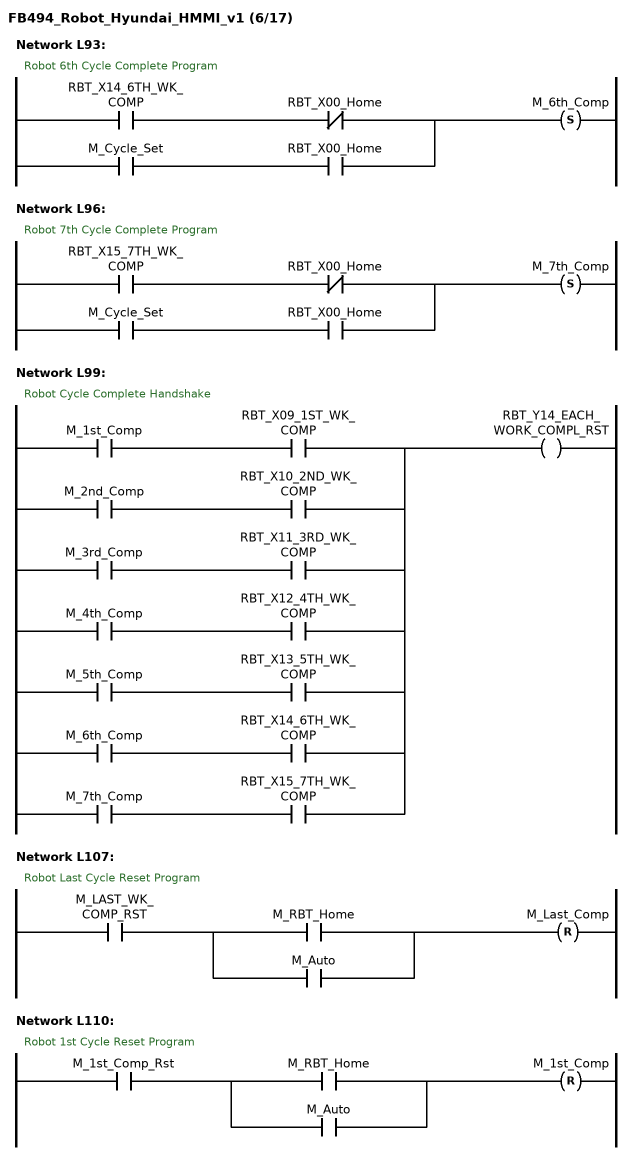
(* [picture p24: FB494_Robot_Hyundai_HMMI_v1 rungs L93-L110] *)
(* Robot 6th Cycle Complete Program *)
(* Rung L93 *)
IF (RBT_X14_6TH_WK_COMP AND NOT RBT_X00_Home) OR (M_Cycle_Set AND RBT_X00_Home) THEN
    M_6th_Comp := TRUE;
END_IF;
(* Robot 7th Cycle Complete Program *)
(* Rung L96 *)
IF (RBT_X15_7TH_WK_COMP AND NOT RBT_X00_Home) OR (M_Cycle_Set AND RBT_X00_Home) THEN
    M_7th_Comp := TRUE;
END_IF;
(* Robot Cycle Complete Handshake *)
(* Rung L99 *)
RBT_Y14_EACH_WORK_COMPL_RST := (M_1st_Comp AND RBT_X09_1ST_WK_COMP) OR (M_2nd_Comp AND RBT_X10_2ND_WK_COMP) OR (M_3rd_Comp AND RBT_X11_3RD_WK_COMP) OR (M_4th_Comp AND RBT_X12_4TH_WK_COMP) OR (M_5th_Comp AND RBT_X13_5TH_WK_COMP) OR (M_6th_Comp AND RBT_X14_6TH_WK_COMP) OR (M_7th_Comp AND RBT_X15_7TH_WK_COMP);
(* Robot Last Cycle Reset Program *)
(* Rung L107 *)
IF M_LAST_WK_COMP_RST AND (M_RBT_Home OR M_Auto) THEN M_Last_Comp := FALSE; END_IF;
(* Robot 1st Cycle Reset Program *)
(* Rung L110 *)
IF M_1st_Comp_Rst AND (M_RBT_Home OR M_Auto) THEN M_1st_Comp := FALSE; END_IF;

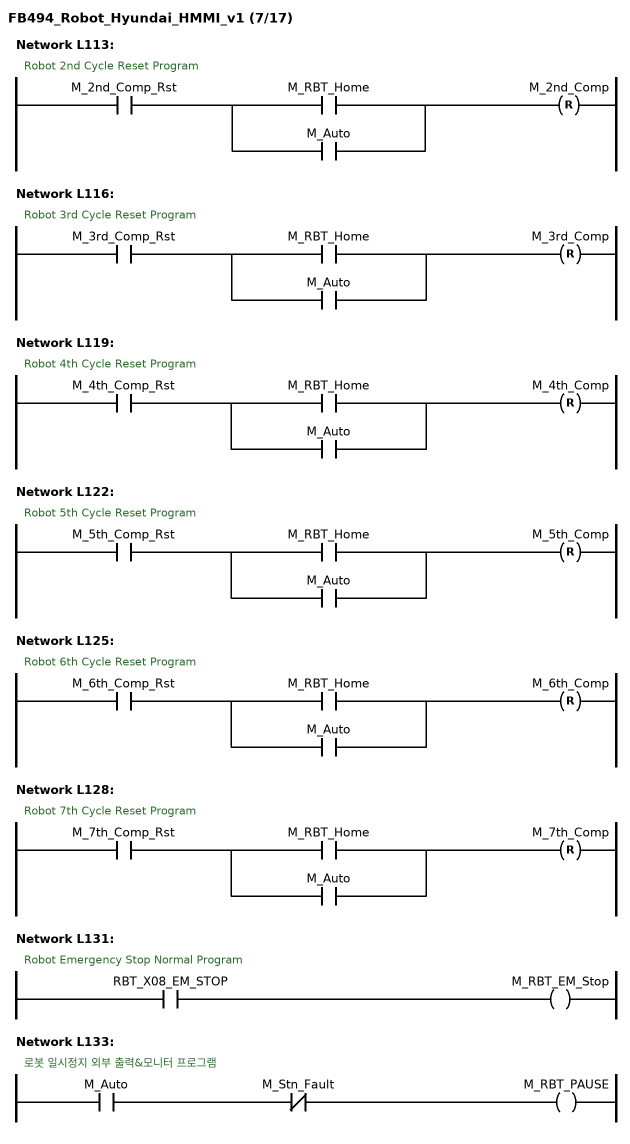
(* Robot 2nd Cycle Reset Program *)
(* Rung L113 *)
IF M_2nd_Comp_Rst AND (M_RBT_Home OR M_Auto) THEN M_2nd_Comp := FALSE; END_IF;
(* Robot 3rd Cycle Reset Program *)
(* Rung L116 *)
IF M_3rd_Comp_Rst AND (M_RBT_Home OR M_Auto) THEN M_3rd_Comp := FALSE; END_IF;
(* Robot 4th Cycle Reset Program *)
(* Rung L119 *)
IF M_4th_Comp_Rst AND (M_RBT_Home OR M_Auto) THEN M_4th_Comp := FALSE; END_IF;
(* Robot 5th Cycle Reset Program *)
(* Rung L122 *)
IF M_5th_Comp_Rst AND (M_RBT_Home OR M_Auto) THEN M_5th_Comp := FALSE; END_IF;
(* Robot 6th Cycle Reset Program *)
(* Rung L125 *)
IF M_6th_Comp_Rst AND (M_RBT_Home OR M_Auto) THEN M_6th_Comp := FALSE; END_IF;
(* Robot 7th Cycle Reset Program *)
(* Rung L128 *)
IF M_7th_Comp_Rst AND (M_RBT_Home OR M_Auto) THEN M_7th_Comp := FALSE; END_IF;
(* Robot Emergency Stop Normal Program *)
(* Rung L131 *)
M_RBT_EM_Stop := RBT_X08_EM_STOP;
(* 로봇 일시정지 외부 출력&모니터 프로그램 *)
(* Rung L133 *)
M_RBT_PAUSE := M_Auto AND NOT M_Stn_Fault;

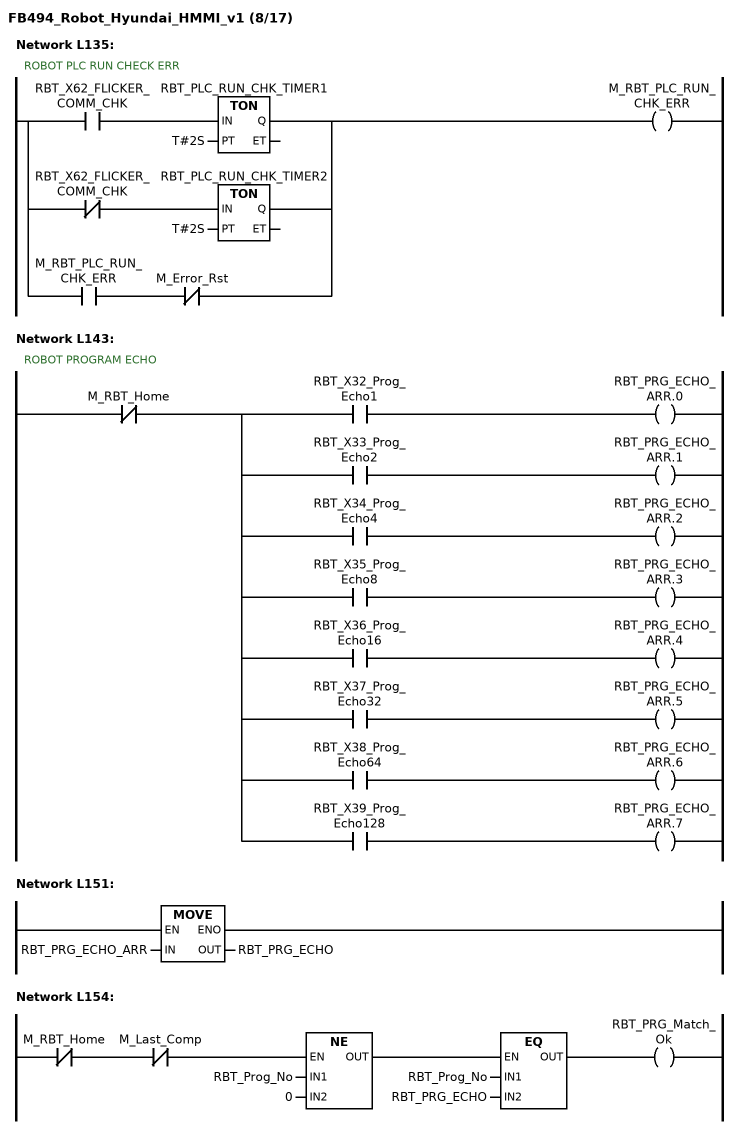
(* ROBOT PLC RUN CHECK ERR *)
(* Rung L135 *)
RBT_PLC_RUN_CHK_TIMER1(IN := RBT_X62_FLICKER_COMM_CHK, PT := T#2S);
RBT_PLC_RUN_CHK_TIMER2(IN := NOT RBT_X62_FLICKER_COMM_CHK, PT := T#2S);
M_RBT_PLC_RUN_CHK_ERR := RBT_PLC_RUN_CHK_TIMER1.Q OR RBT_PLC_RUN_CHK_TIMER2.Q OR (M_RBT_PLC_RUN_CHK_ERR AND NOT M_Error_Rst);
(* ROBOT PROGRAM ECHO *)
(* Rung L143 *)
RBT_PRG_ECHO_ARR.0 := NOT M_RBT_Home AND RBT_X32_Prog_Echo1;
RBT_PRG_ECHO_ARR.1 := NOT M_RBT_Home AND RBT_X33_Prog_Echo2;
RBT_PRG_ECHO_ARR.2 := NOT M_RBT_Home AND RBT_X34_Prog_Echo4;
RBT_PRG_ECHO_ARR.3 := NOT M_RBT_Home AND RBT_X35_Prog_Echo8;
RBT_PRG_ECHO_ARR.4 := NOT M_RBT_Home AND RBT_X36_Prog_Echo16;
RBT_PRG_ECHO_ARR.5 := NOT M_RBT_Home AND RBT_X37_Prog_Echo32;
RBT_PRG_ECHO_ARR.6 := NOT M_RBT_Home AND RBT_X38_Prog_Echo64;
RBT_PRG_ECHO_ARR.7 := NOT M_RBT_Home AND RBT_X39_Prog_Echo128;
(* Rung L151 *)
RBT_PRG_ECHO := RBT_PRG_ECHO_ARR;
(* Rung L154 *)
IF NOT M_RBT_Home AND NOT M_Last_Comp THEN _t1 := RBT_Prog_No <> 0; END_IF;
IF _t1 THEN _t2 := RBT_Prog_No = RBT_PRG_ECHO; END_IF;
RBT_PRG_Match_Ok := _t2;

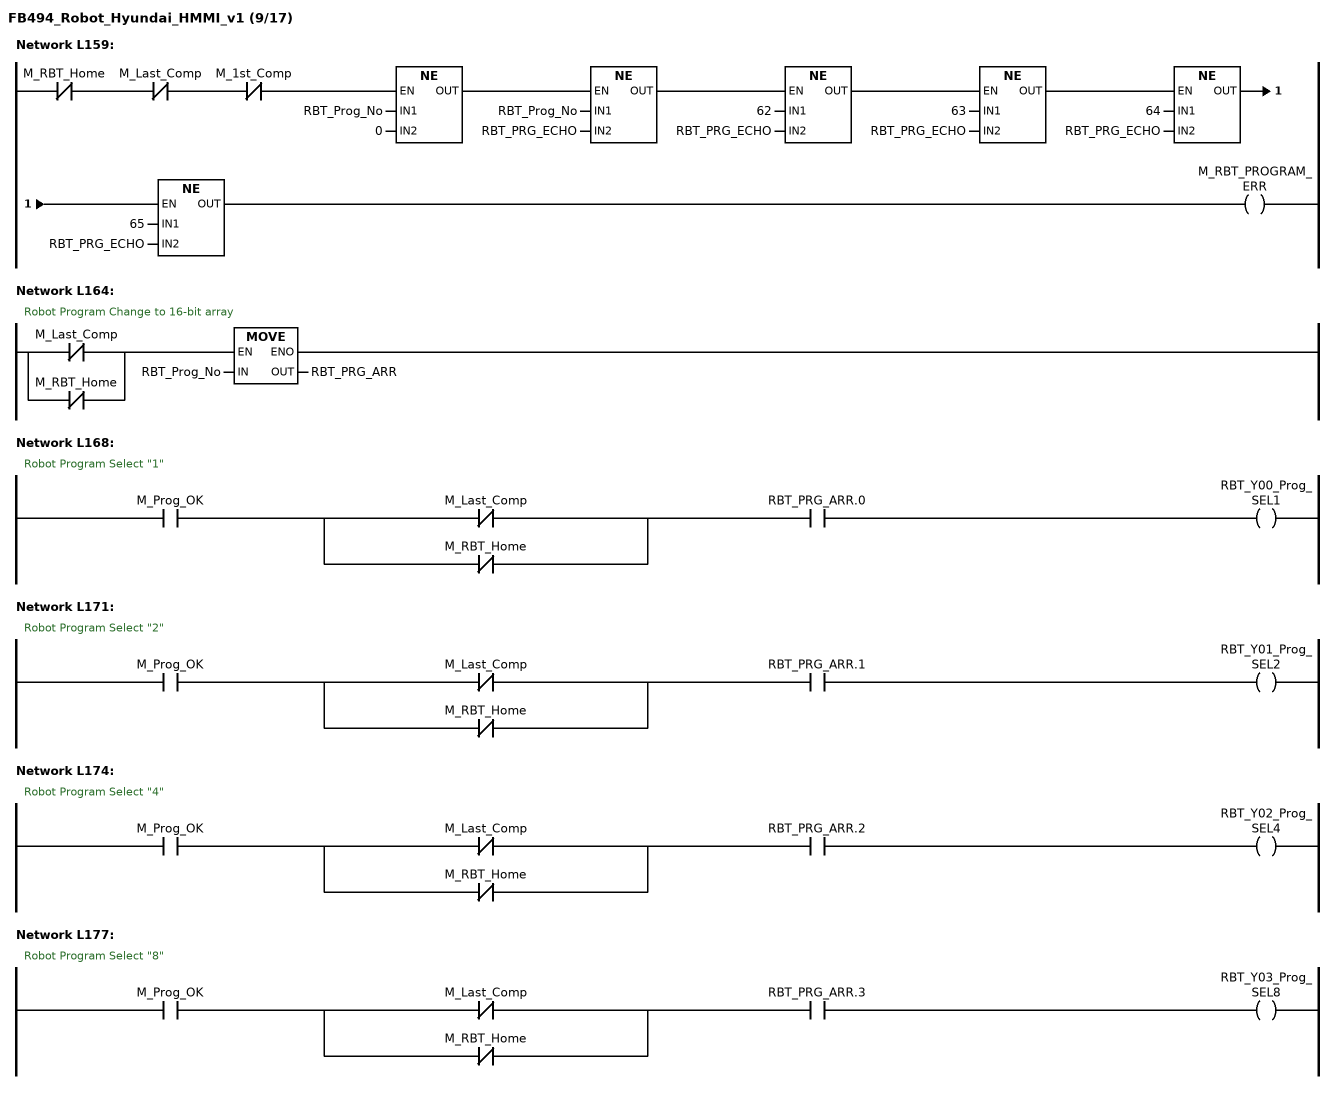
(* Rung L159 *)
IF NOT M_RBT_Home AND NOT M_Last_Comp AND NOT M_1st_Comp THEN _t3 := RBT_Prog_No <> 0; END_IF;
IF _t3 THEN _t4 := RBT_Prog_No <> RBT_PRG_ECHO; END_IF;
IF _t4 THEN _t5 := 62 <> RBT_PRG_ECHO; END_IF;
IF _t5 THEN _t6 := 63 <> RBT_PRG_ECHO; END_IF;
IF _t6 THEN _t7 := 64 <> RBT_PRG_ECHO; END_IF;
IF _t7 THEN _t8 := 65 <> RBT_PRG_ECHO; END_IF;
M_RBT_PROGRAM_ERR := _t8;
(* Robot Program Change to 16-bit array *)
(* Rung L164 *)
IF NOT M_Last_Comp OR NOT M_RBT_Home THEN RBT_PRG_ARR := RBT_Prog_No; END_IF;
(* Robot Program Select "1" *)
(* Rung L168 *)
RBT_Y00_Prog_SEL1 := M_Prog_OK AND (NOT M_Last_Comp OR NOT M_RBT_Home) AND RBT_PRG_ARR.0;
(* Robot Program Select "2" *)
(* Rung L171 *)
RBT_Y01_Prog_SEL2 := M_Prog_OK AND (NOT M_Last_Comp OR NOT M_RBT_Home) AND RBT_PRG_ARR.1;
(* Robot Program Select "4" *)
(* Rung L174 *)
RBT_Y02_Prog_SEL4 := M_Prog_OK AND (NOT M_Last_Comp OR NOT M_RBT_Home) AND RBT_PRG_ARR.2;
(* Robot Program Select "8" *)
(* Rung L177 *)
RBT_Y03_Prog_SEL8 := M_Prog_OK AND (NOT M_Last_Comp OR NOT M_RBT_Home) AND RBT_PRG_ARR.3;

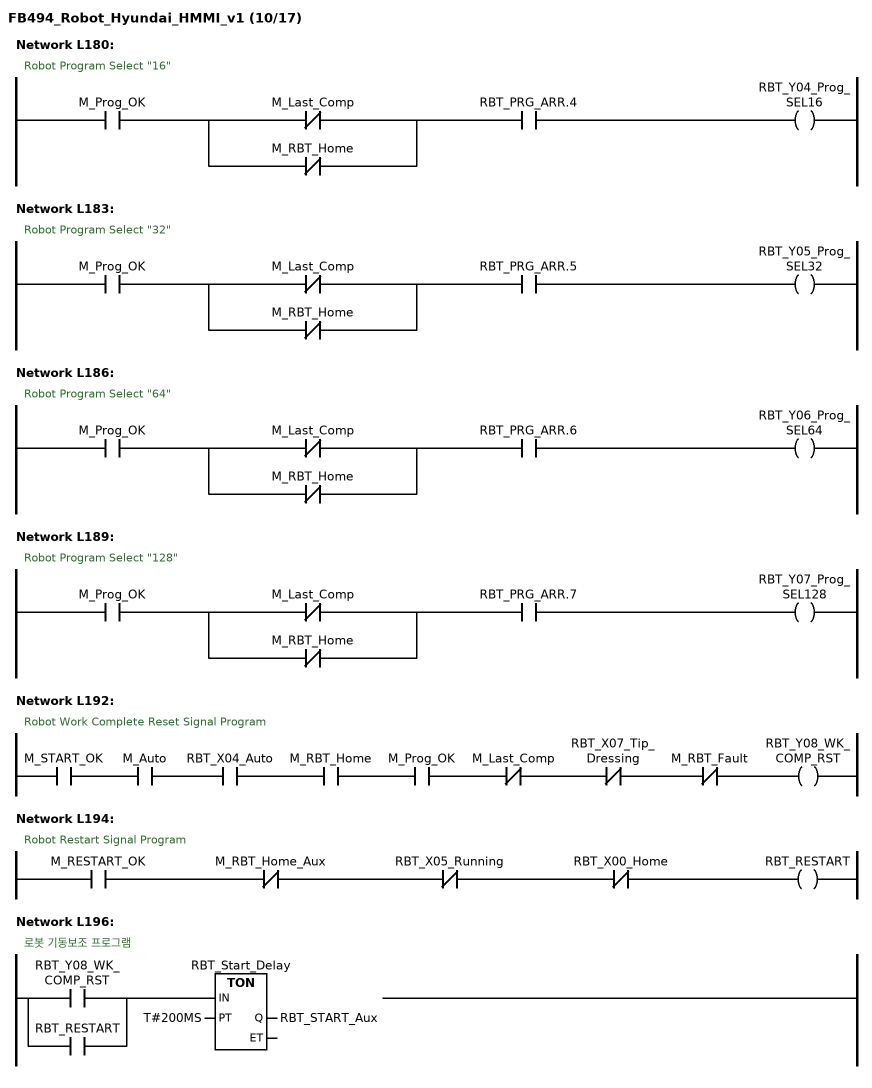
(* Robot Program Select "16" *)
(* Rung L180 *)
RBT_Y04_Prog_SEL16 := M_Prog_OK AND (NOT M_Last_Comp OR NOT M_RBT_Home) AND RBT_PRG_ARR.4;
(* Robot Program Select "32" *)
(* Rung L183 *)
RBT_Y05_Prog_SEL32 := M_Prog_OK AND (NOT M_Last_Comp OR NOT M_RBT_Home) AND RBT_PRG_ARR.5;
(* Robot Program Select "64" *)
(* Rung L186 *)
RBT_Y06_Prog_SEL64 := M_Prog_OK AND (NOT M_Last_Comp OR NOT M_RBT_Home) AND RBT_PRG_ARR.6;
(* Robot Program Select "128" *)
(* Rung L189 *)
RBT_Y07_Prog_SEL128 := M_Prog_OK AND (NOT M_Last_Comp OR NOT M_RBT_Home) AND RBT_PRG_ARR.7;
(* Robot Work Complete Reset Signal Program *)
(* Rung L192 *)
RBT_Y08_WK_COMP_RST := M_START_OK AND M_Auto AND RBT_X04_Auto AND M_RBT_Home AND M_Prog_OK AND NOT M_Last_Comp AND NOT RBT_X07_Tip_Dressing AND NOT M_RBT_Fault;
(* Robot Restart Signal Program *)
(* Rung L194 *)
RBT_RESTART := M_RESTART_OK AND NOT M_RBT_Home_Aux AND NOT RBT_X05_Running AND NOT RBT_X00_Home;
(* 로봇 기동보조 프로그램 *)
(* Rung L196 *)
RBT_Start_Delay(IN := RBT_Y08_WK_COMP_RST OR RBT_RESTART, PT := T#200MS, Q => RBT_START_Aux);

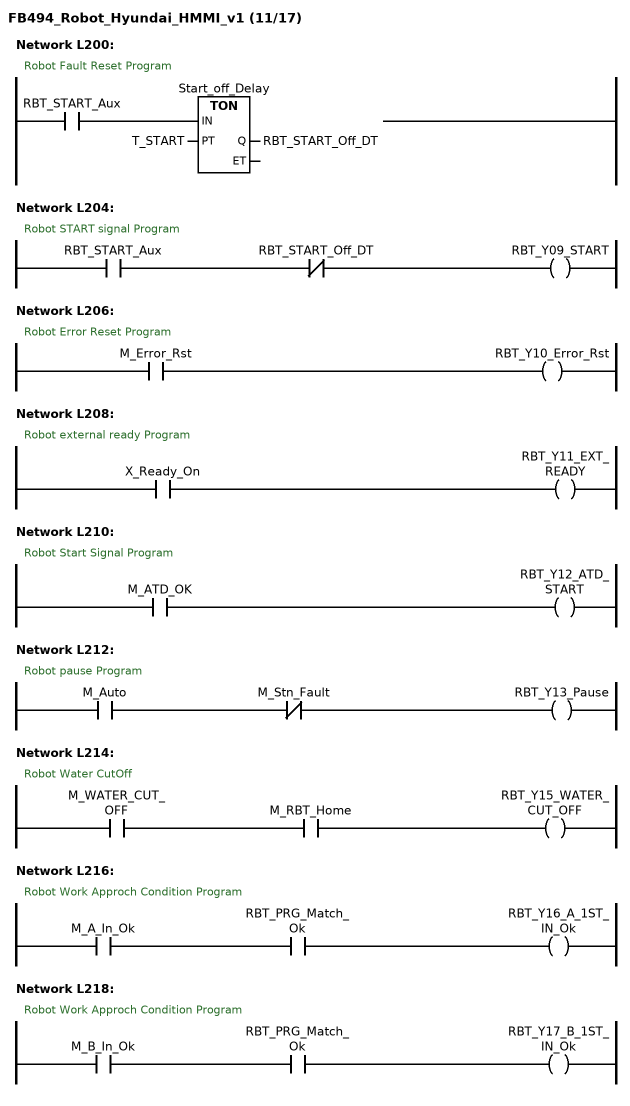
(* Robot Fault Reset Program *)
(* Rung L200 *)
Start_off_Delay(IN := RBT_START_Aux, PT := T_START, Q => RBT_START_Off_DT);
(* Robot START signal Program *)
(* Rung L204 *)
RBT_Y09_START := RBT_START_Aux AND NOT RBT_START_Off_DT;
(* Robot Error Reset Program *)
(* Rung L206 *)
RBT_Y10_Error_Rst := M_Error_Rst;
(* Robot external ready Program *)
(* Rung L208 *)
RBT_Y11_EXT_READY := X_Ready_On;
(* Robot Start Signal Program *)
(* Rung L210 *)
RBT_Y12_ATD_START := M_ATD_OK;
(* Robot pause Program *)
(* Rung L212 *)
RBT_Y13_Pause := M_Auto AND NOT M_Stn_Fault;
(* Robot Water CutOff *)
(* Rung L214 *)
RBT_Y15_WATER_CUT_OFF := M_WATER_CUT_OFF AND M_RBT_Home;
(* Robot Work Approch Condition Program *)
(* Rung L216 *)
RBT_Y16_A_1ST_IN_Ok := M_A_In_Ok AND RBT_PRG_Match_Ok;
(* Robot Work Approch Condition Program *)
(* Rung L218 *)
RBT_Y17_B_1ST_IN_Ok := M_B_In_Ok AND RBT_PRG_Match_Ok;

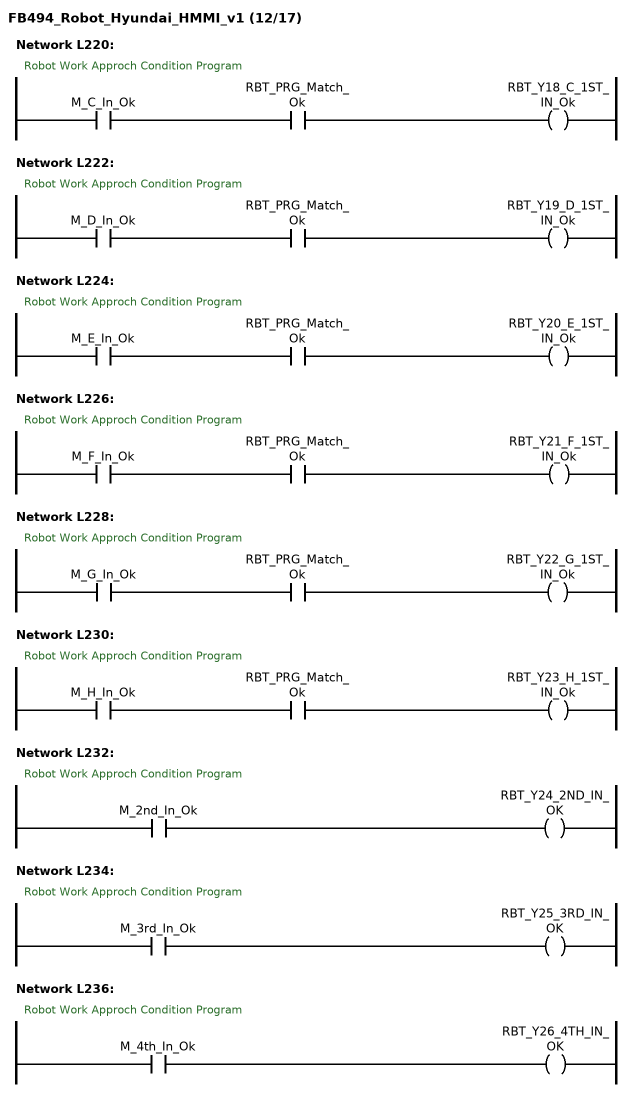
(* Robot Work Approch Condition Program *)
(* Rung L220 *)
RBT_Y18_C_1ST_IN_Ok := M_C_In_Ok AND RBT_PRG_Match_Ok;
(* Robot Work Approch Condition Program *)
(* Rung L222 *)
RBT_Y19_D_1ST_IN_Ok := M_D_In_Ok AND RBT_PRG_Match_Ok;
(* Robot Work Approch Condition Program *)
(* Rung L224 *)
RBT_Y20_E_1ST_IN_Ok := M_E_In_Ok AND RBT_PRG_Match_Ok;
(* Robot Work Approch Condition Program *)
(* Rung L226 *)
RBT_Y21_F_1ST_IN_Ok := M_F_In_Ok AND RBT_PRG_Match_Ok;
(* Robot Work Approch Condition Program *)
(* Rung L228 *)
RBT_Y22_G_1ST_IN_Ok := M_G_In_Ok AND RBT_PRG_Match_Ok;
(* Robot Work Approch Condition Program *)
(* Rung L230 *)
RBT_Y23_H_1ST_IN_Ok := M_H_In_Ok AND RBT_PRG_Match_Ok;
(* Robot Work Approch Condition Program *)
(* Rung L232 *)
RBT_Y24_2ND_IN_OK := M_2nd_In_Ok;
(* Robot Work Approch Condition Program *)
(* Rung L234 *)
RBT_Y25_3RD_IN_OK := M_3rd_In_Ok;
(* Robot Work Approch Condition Program *)
(* Rung L236 *)
RBT_Y26_4TH_IN_OK := M_4th_In_Ok;

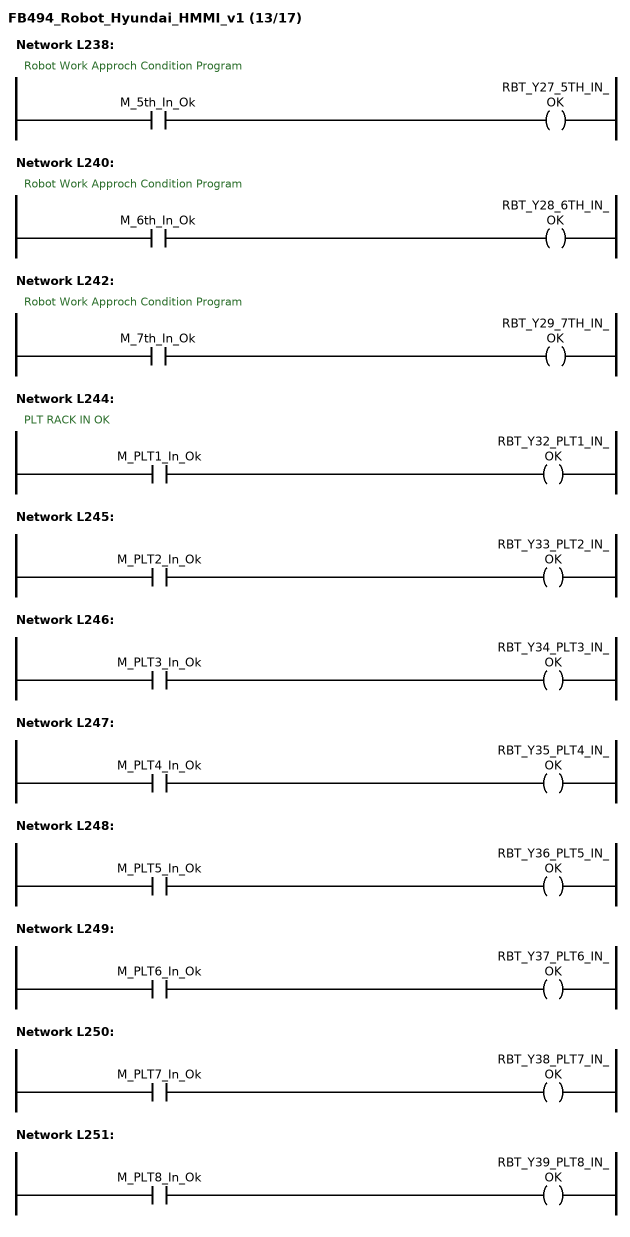
(* Robot Work Approch Condition Program *)
(* Rung L238 *)
RBT_Y27_5TH_IN_OK := M_5th_In_Ok;
(* Robot Work Approch Condition Program *)
(* Rung L240 *)
RBT_Y28_6TH_IN_OK := M_6th_In_Ok;
(* Robot Work Approch Condition Program *)
(* Rung L242 *)
RBT_Y29_7TH_IN_OK := M_7th_In_Ok;
(* PLT RACK IN OK *)
(* Rung L244 *)
RBT_Y32_PLT1_IN_OK := M_PLT1_In_Ok;
(* Rung L245 *)
RBT_Y33_PLT2_IN_OK := M_PLT2_In_Ok;
(* Rung L246 *)
RBT_Y34_PLT3_IN_OK := M_PLT3_In_Ok;
(* Rung L247 *)
RBT_Y35_PLT4_IN_OK := M_PLT4_In_Ok;
(* Rung L248 *)
RBT_Y36_PLT5_IN_OK := M_PLT5_In_Ok;
(* Rung L249 *)
RBT_Y37_PLT6_IN_OK := M_PLT6_In_Ok;
(* Rung L250 *)
RBT_Y38_PLT7_IN_OK := M_PLT7_In_Ok;
(* Rung L251 *)
RBT_Y39_PLT8_IN_OK := M_PLT8_In_Ok;

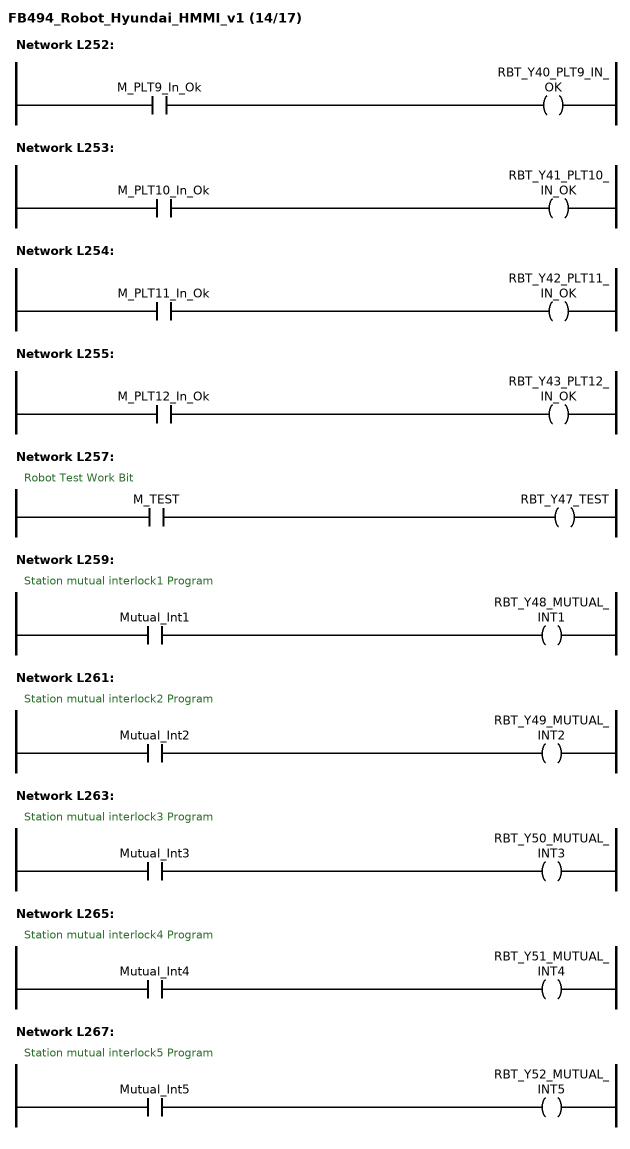
(* Rung L252 *)
RBT_Y40_PLT9_IN_OK := M_PLT9_In_Ok;
(* Rung L253 *)
RBT_Y41_PLT10_IN_OK := M_PLT10_In_Ok;
(* Rung L254 *)
RBT_Y42_PLT11_IN_OK := M_PLT11_In_Ok;
(* Rung L255 *)
RBT_Y43_PLT12_IN_OK := M_PLT12_In_Ok;
(* Robot Test Work Bit *)
(* Rung L257 *)
RBT_Y47_TEST := M_TEST;
(* Station mutual interlock1 Program *)
(* Rung L259 *)
RBT_Y48_MUTUAL_INT1 := Mutual_Int1;
(* Station mutual interlock2 Program *)
(* Rung L261 *)
RBT_Y49_MUTUAL_INT2 := Mutual_Int2;
(* Station mutual interlock3 Program *)
(* Rung L263 *)
RBT_Y50_MUTUAL_INT3 := Mutual_Int3;
(* Station mutual interlock4 Program *)
(* Rung L265 *)
RBT_Y51_MUTUAL_INT4 := Mutual_Int4;
(* Station mutual interlock5 Program *)
(* Rung L267 *)
RBT_Y52_MUTUAL_INT5 := Mutual_Int5;

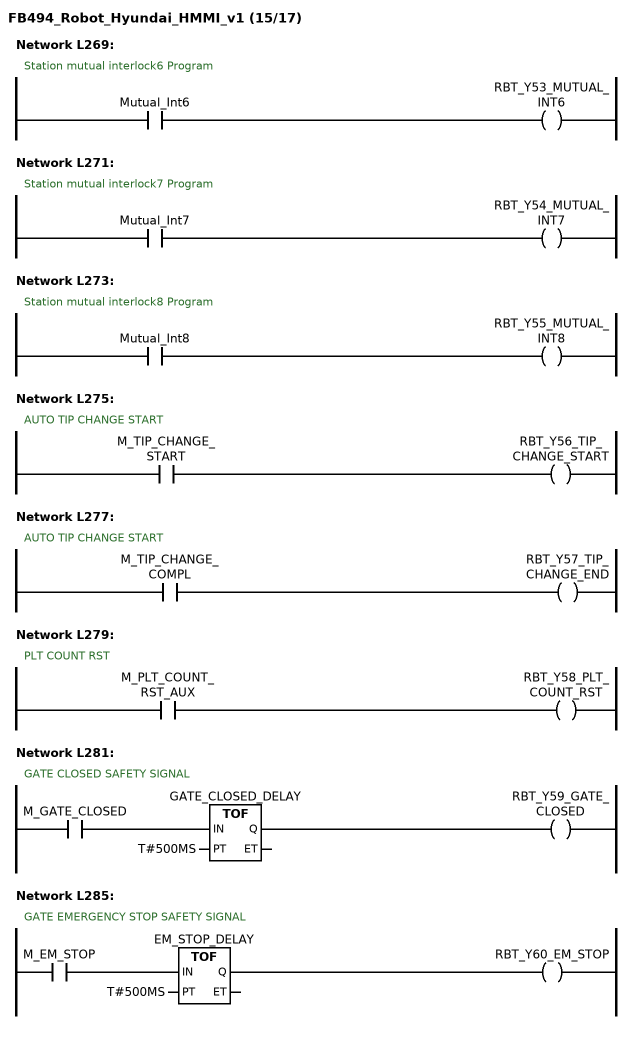
(* Station mutual interlock6 Program *)
(* Rung L269 *)
RBT_Y53_MUTUAL_INT6 := Mutual_Int6;
(* Station mutual interlock7 Program *)
(* Rung L271 *)
RBT_Y54_MUTUAL_INT7 := Mutual_Int7;
(* Station mutual interlock8 Program *)
(* Rung L273 *)
RBT_Y55_MUTUAL_INT8 := Mutual_Int8;
(* AUTO TIP CHANGE START *)
(* Rung L275 *)
RBT_Y56_TIP_CHANGE_START := M_TIP_CHANGE_START;
(* AUTO TIP CHANGE START *)
(* Rung L277 *)
RBT_Y57_TIP_CHANGE_END := M_TIP_CHANGE_COMPL;
(* PLT COUNT RST *)
(* Rung L279 *)
RBT_Y58_PLT_COUNT_RST := M_PLT_COUNT_RST_AUX;
(* GATE CLOSED SAFETY SIGNAL *)
(* Rung L281 *)
GATE_CLOSED_DELAY(IN := M_GATE_CLOSED, PT := T#500MS);
RBT_Y59_GATE_CLOSED := GATE_CLOSED_DELAY.Q;
(* GATE EMERGENCY STOP SAFETY SIGNAL *)
(* Rung L285 *)
EM_STOP_DELAY(IN := M_EM_STOP, PT := T#500MS);
RBT_Y60_EM_STOP := EM_STOP_DELAY.Q;

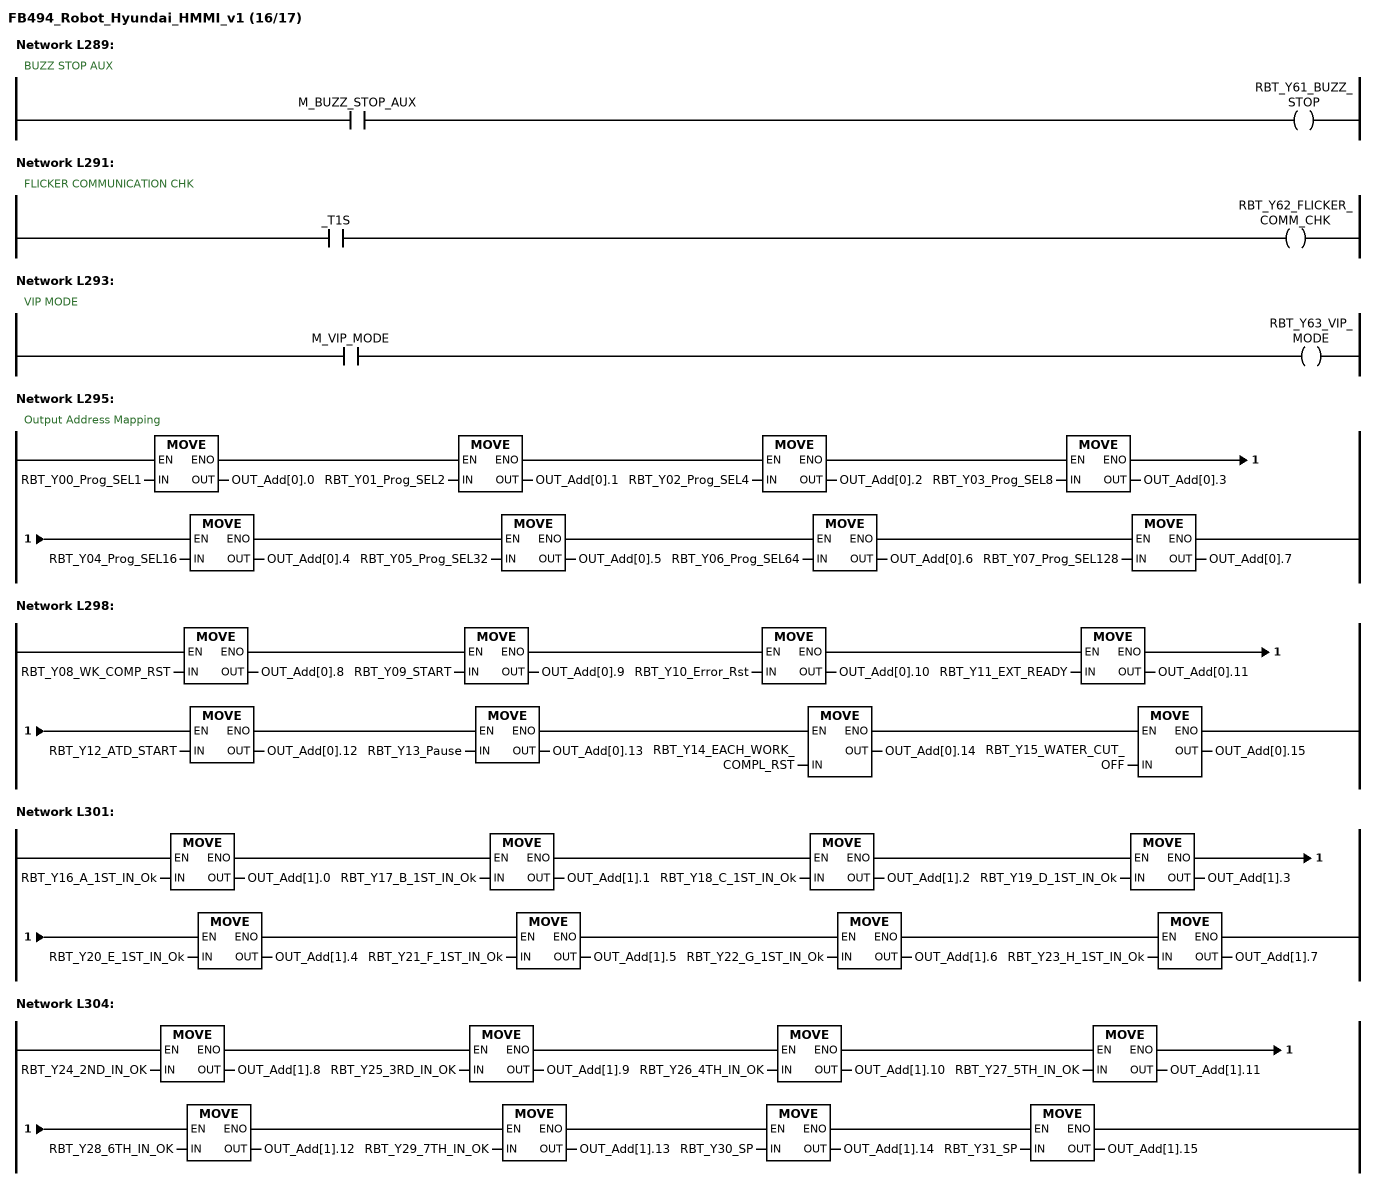
(* BUZZ STOP AUX *)
(* Rung L289 *)
RBT_Y61_BUZZ_STOP := M_BUZZ_STOP_AUX;
(* FLICKER COMMUNICATION CHK *)
(* Rung L291 *)
RBT_Y62_FLICKER_COMM_CHK := _T1S;
(* VIP MODE *)
(* Rung L293 *)
RBT_Y63_VIP_MODE := M_VIP_MODE;
(* Output Address Mapping *)
(* Rung L295 *)
OUT_Add[0].0 := RBT_Y00_Prog_SEL1;
OUT_Add[0].1 := RBT_Y01_Prog_SEL2;
OUT_Add[0].2 := RBT_Y02_Prog_SEL4;
OUT_Add[0].3 := RBT_Y03_Prog_SEL8;
OUT_Add[0].4 := RBT_Y04_Prog_SEL16;
OUT_Add[0].5 := RBT_Y05_Prog_SEL32;
OUT_Add[0].6 := RBT_Y06_Prog_SEL64;
OUT_Add[0].7 := RBT_Y07_Prog_SEL128;
(* Rung L298 *)
OUT_Add[0].8 := RBT_Y08_WK_COMP_RST;
OUT_Add[0].9 := RBT_Y09_START;
OUT_Add[0].10 := RBT_Y10_Error_Rst;
OUT_Add[0].11 := RBT_Y11_EXT_READY;
OUT_Add[0].12 := RBT_Y12_ATD_START;
OUT_Add[0].13 := RBT_Y13_Pause;
OUT_Add[0].14 := RBT_Y14_EACH_WORK_COMPL_RST;
OUT_Add[0].15 := RBT_Y15_WATER_CUT_OFF;
(* Rung L301 *)
OUT_Add[1].0 := RBT_Y16_A_1ST_IN_Ok;
OUT_Add[1].1 := RBT_Y17_B_1ST_IN_Ok;
OUT_Add[1].2 := RBT_Y18_C_1ST_IN_Ok;
OUT_Add[1].3 := RBT_Y19_D_1ST_IN_Ok;
OUT_Add[1].4 := RBT_Y20_E_1ST_IN_Ok;
OUT_Add[1].5 := RBT_Y21_F_1ST_IN_Ok;
OUT_Add[1].6 := RBT_Y22_G_1ST_IN_Ok;
OUT_Add[1].7 := RBT_Y23_H_1ST_IN_Ok;
(* Rung L304 *)
OUT_Add[1].8 := RBT_Y24_2ND_IN_OK;
OUT_Add[1].9 := RBT_Y25_3RD_IN_OK;
OUT_Add[1].10 := RBT_Y26_4TH_IN_OK;
OUT_Add[1].11 := RBT_Y27_5TH_IN_OK;
OUT_Add[1].12 := RBT_Y28_6TH_IN_OK;
OUT_Add[1].13 := RBT_Y29_7TH_IN_OK;
OUT_Add[1].14 := RBT_Y30_SP;
OUT_Add[1].15 := RBT_Y31_SP;

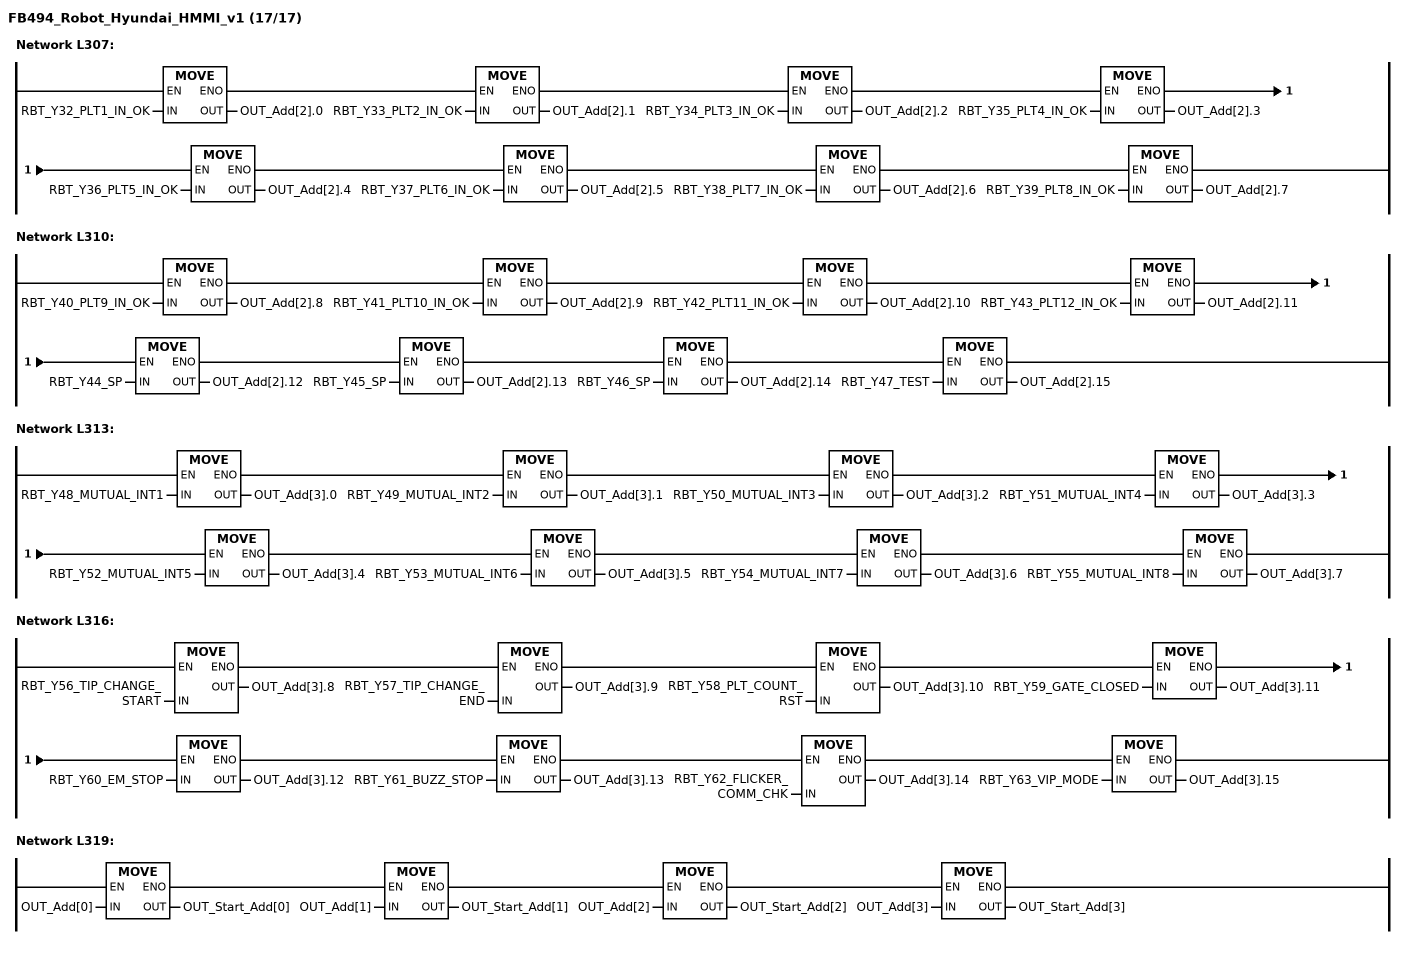
(* Rung L307 *)
OUT_Add[2].0 := RBT_Y32_PLT1_IN_OK;
OUT_Add[2].1 := RBT_Y33_PLT2_IN_OK;
OUT_Add[2].2 := RBT_Y34_PLT3_IN_OK;
OUT_Add[2].3 := RBT_Y35_PLT4_IN_OK;
OUT_Add[2].4 := RBT_Y36_PLT5_IN_OK;
OUT_Add[2].5 := RBT_Y37_PLT6_IN_OK;
OUT_Add[2].6 := RBT_Y38_PLT7_IN_OK;
OUT_Add[2].7 := RBT_Y39_PLT8_IN_OK;
(* Rung L310 *)
OUT_Add[2].8 := RBT_Y40_PLT9_IN_OK;
OUT_Add[2].9 := RBT_Y41_PLT10_IN_OK;
OUT_Add[2].10 := RBT_Y42_PLT11_IN_OK;
OUT_Add[2].11 := RBT_Y43_PLT12_IN_OK;
OUT_Add[2].12 := RBT_Y44_SP;
OUT_Add[2].13 := RBT_Y45_SP;
OUT_Add[2].14 := RBT_Y46_SP;
OUT_Add[2].15 := RBT_Y47_TEST;
(* Rung L313 *)
OUT_Add[3].0 := RBT_Y48_MUTUAL_INT1;
OUT_Add[3].1 := RBT_Y49_MUTUAL_INT2;
OUT_Add[3].2 := RBT_Y50_MUTUAL_INT3;
OUT_Add[3].3 := RBT_Y51_MUTUAL_INT4;
OUT_Add[3].4 := RBT_Y52_MUTUAL_INT5;
OUT_Add[3].5 := RBT_Y53_MUTUAL_INT6;
OUT_Add[3].6 := RBT_Y54_MUTUAL_INT7;
OUT_Add[3].7 := RBT_Y55_MUTUAL_INT8;
(* Rung L316 *)
OUT_Add[3].8 := RBT_Y56_TIP_CHANGE_START;
OUT_Add[3].9 := RBT_Y57_TIP_CHANGE_END;
OUT_Add[3].10 := RBT_Y58_PLT_COUNT_RST;
OUT_Add[3].11 := RBT_Y59_GATE_CLOSED;
OUT_Add[3].12 := RBT_Y60_EM_STOP;
OUT_Add[3].13 := RBT_Y61_BUZZ_STOP;
OUT_Add[3].14 := RBT_Y62_FLICKER_COMM_CHK;
OUT_Add[3].15 := RBT_Y63_VIP_MODE;
(* Rung L319 *)
OUT_Start_Add[0] := OUT_Add[0];
OUT_Start_Add[1] := OUT_Add[1];
OUT_Start_Add[2] := OUT_Add[2];
OUT_Start_Add[3] := OUT_Add[3];
END_FUNCTION_BLOCK

PROGRAM MCP_유틸리티 (* task: 스캔 프로그램 *)
VAR_EXTERNAL RETAIN
    ALWAYS_ON : BOOL; (* AT %MW3.1 *) (* 항시 ON *)
    CLOCK_BIT_1_0Sec : BOOL; (* AT %MW0.5 *) (* CLOCK_BIT_1_0Sec *)
    GATE1_M_이상_리셋 : BOOL; (* AT %MW400.0 *) (* GATE1 PB 이상리셋 *)
    GATE2_M_이상_리셋 : BOOL; (* AT %MW401.0 *) (* GATE2 PB 이상리셋 *)
    GATE3_M_이상_리셋 : BOOL; (* AT %MW402.0 *) (* GATE3 PB 이상리셋 *)
    HOP1_M_부저_정지 : BOOL; (* AT %MW360.5 *) (* HOP1 PB 부저정지 *)
    HOP1_M_비상정지 : BOOL; (* AT %MW360.7 *) (* HOP1 비상정지 이상 *)
    HOP1_M_이상_리셋 : BOOL; (* AT %MW360.4 *) (* HOP1 PB 이상리셋 *)
    MCP_M_램프_테스트 : BOOL; (* AT %MW350.6 *) (* MCP SPB LAMP 테스트 *)
    MCP_M_부저_정지 : BOOL; (* AT %MW350.5 *) (* MCP 부저정지 *)
    MCP_M_비상정지 : BOOL; (* AT %MW350.7 *) (* MCP 비상정지 이상 *)
    MCP_M_수동모드 : BOOL; (* AT %MW350.1 *) (* MCP ALL공정 수동모드 *)
    MCP_M_운전준비_ON : BOOL; (* AT %MW350.0 *) (* MCP ALL공정 운전준비 ON *)
    MCP_M_이상_리셋 : BOOL; (* AT %MW350.4 *) (* MCP PB 이상리셋 *)
    MCP_M_자동_운전중 : BOOL; (* AT %MW350.3 *) (* MCP ALL공정 자동운전중 *)
    MCP_M_자동모드 : BOOL; (* AT %MW350.2 *) (* MCP ALL공정 자동모드 *)
    S362_M_수동모드 : BOOL; (* AT %MW1000.3 *) (* S362 선택 수동모드 *)
    S362_M_운전준비_ON : BOOL; (* AT %MW1000.0 *) (* S362 운전준비 ON *)
    S362_M_자동_START : BOOL; (* AT %MW1000.5 *) (* S362 자동운전중 *)
    S362_M_자동_운전중 : BOOL; (* AT %MW1000.4 *) (* S362 자동운전중 *)
    S362_M_자동모드 : BOOL; (* AT %MW1000.1 *) (* S362 선택 자동모드 *)
    S364_M_수동모드 : BOOL; (* AT %MW2000.3 *) (* S364 선택 수동모드 *)
    S364_M_운전준비_ON : BOOL; (* AT %MW2000.0 *) (* S364 운전준비 ON *)
    S364_M_자동_START : BOOL; (* AT %MW2000.5 *) (* S364 자동운전중 *)
    S364_M_자동_운전중 : BOOL; (* AT %MW2000.4 *) (* S364 자동운전중 *)
    S364_M_자동모드 : BOOL; (* AT %MW2000.1 *) (* S364 선택 자동모드 *)
    S365_M_수동모드 : BOOL; (* AT %MW2500.3 *) (* S365 선택 수동모드 *)
    S365_M_운전준비_ON : BOOL; (* AT %MW2500.0 *) (* S365 운전준비 ON *)
    S365_M_자동_START : BOOL; (* AT %MW2500.5 *) (* S365 자동운전중 *)
    S365_M_자동_운전중 : BOOL; (* AT %MW2500.4 *) (* S365 자동운전중 *)
    S365_M_자동모드 : BOOL; (* AT %MW2500.1 *) (* S365 선택 자동모드 *)
    S366_M_수동모드 : BOOL; (* AT %MW3000.3 *) (* S366 선택 수동모드 *)
    S366_M_운전준비_ON : BOOL; (* AT %MW3000.0 *) (* S366 운전준비 ON *)
    S366_M_자동_START : BOOL; (* AT %MW3000.5 *) (* S366 자동운전중 *)
    S366_M_자동_운전중 : BOOL; (* AT %MW3000.4 *) (* S366 자동운전중 *)
    S366_M_자동모드 : BOOL; (* AT %MW3000.1 *) (* S366 선택 자동모드 *)
    S367_M_수동모드 : BOOL; (* AT %MW3500.3 *) (* S367 선택 수동모드 *)
    S367_M_운전준비_ON : BOOL; (* AT %MW3500.0 *) (* S367 운전준비 ON *)
    S367_M_자동_START : BOOL; (* AT %MW3500.5 *) (* S367 자동운전중 *)
    S367_M_자동_운전중 : BOOL; (* AT %MW3500.4 *) (* S367 자동운전중 *)
    S367_M_자동모드 : BOOL; (* AT %MW3500.1 *) (* S367 선택 자동모드 *)
    S368_M_수동모드 : BOOL; (* AT %MW4000.3 *) (* S368 선택 수동모드 *)
    S368_M_운전준비_ON : BOOL; (* AT %MW4000.0 *) (* S368 운전준비 ON *)
    S368_M_자동_START : BOOL; (* AT %MW4000.5 *) (* S368 자동운전중 *)
    S368_M_자동_운전중 : BOOL; (* AT %MW4000.4 *) (* S368 자동운전중 *)
    S368_M_자동모드 : BOOL; (* AT %MW4000.1 *) (* S368 선택 자동모드 *)
    S369_1_M_수동모드 : BOOL; (* AT %MW4500.3 *) (* S369-1 선택 수동모드 *)
    S369_1_M_운전준비_ON : BOOL; (* AT %MW4500.0 *) (* S369-1 운전준비 ON *)
    S369_1_M_자동_START : BOOL; (* AT %MW4500.5 *) (* S369-1 자동운전중 *)
    S369_1_M_자동_운전중 : BOOL; (* AT %MW4500.4 *) (* S369-1 자동운전중 *)
    S369_1_M_자동모드 : BOOL; (* AT %MW4500.1 *) (* S369-1 선택 자동모드 *)
    S369_M_수동모드 : BOOL; (* AT %MW5000.3 *) (* S369 선택 수동모드 *)
    S369_M_운전준비_ON : BOOL; (* AT %MW5000.0 *) (* S369 운전준비 ON *)
    S369_M_자동_START : BOOL; (* AT %MW5000.5 *) (* S369 자동운전중 *)
    S369_M_자동_운전중 : BOOL; (* AT %MW5000.4 *) (* S369 자동운전중 *)
    S369_M_자동모드 : BOOL; (* AT %MW5000.1 *) (* S369 선택 자동모드 *)
    전체_M_운전준비_보조 : BOOL; (* AT %MW308.5 *)
    전체_M_이상_리셋 : BOOL; (* AT %MW308.2 *) (* ALL공정 PB 이상리셋 *)
    전체_라인_M_총괄_GATE_OPEN_이상 : BOOL; (* AT %MW301.5 *) (* ALL공정 GATEBOX 이상총괄 *)
    전체_라인_M_총괄_ROBOT_이상 : BOOL; (* AT %MW301.1 *) (* ALL공정 ROBOT 총괄이상 *)
    전체_라인_M_총괄_SAFETY_이상 : BOOL; (* AT %MW300.2 *) (* ALL공정 SAFETY  이상총괄 *)
    전체_라인_M_총괄_비상정지_이상 : BOOL; (* AT %MW300.1 *) (* ALL공정 비상정지 이상총괄 *)
    전체_라인_M_총괄_이상 : BOOL; (* AT %MW300.0 *) (* ALL공정 총괄이상 *)
END_VAR
VAR_EXTERNAL
    EGIS_CWS : BOOL;
    EGIS_ON : BOOL; (* 항시ON (임시용) *)
    HOP_PBL_운전준비_ON : BOOL; (* AT %MW87500.0 *) (* HOP_PBL_운전준비_ON *)
    MCP_EPB_비상정지1 : BOOL; (* AT %MW87635.0 *) (* MCP_EPB_비상정지1 *)
    MCP_EPB_비상정지2 : BOOL; (* AT %MW87635.1 *) (* MCP_EPB_비상정지2 *)
    MCP_PBL_362_4_자동_운전 : BOOL; (* AT %MW87630.4 *) (* MCP PBL 362~4 자동기동 *)
    MCP_PBL_362_4_자동_운전_LP : BOOL; (* AT %MW97633.1 *) (* MCP PBL 362~4 자동운전중 (램프) *)
    MCP_PBL_365_8_자동_운전 : BOOL; (* AT %MW87630.7 *) (* MCP PBL 365~8 자동기동 *)
    MCP_PBL_365_8_자동_운전_LP : BOOL; (* AT %MW97633.2 *) (* MCP PBL 365~8 자동운전중 (램프) *)
    MCP_PBL_369_자동_운전 : BOOL; (* AT %MW87630.10 *) (* MCP PBL 369~-1 자동기동 *)
    MCP_PBL_369_자동_운전_LP : BOOL; (* AT %MW97633.3 *) (* MCP PBL 369~-1 자동운전중 (램프) *)
    MCP_PBL_운전준비_ON : BOOL; (* AT %MW87630.0 *) (* MCP_PBL_운전준비_ON *)
    MCP_PBL_운전준비_ON_LP : BOOL; (* AT %MW97633.0 *) (* MCP PBL 운전준비ON (램프) *)
    MCP_PB_이상_리셋 : BOOL; (* AT %MW87630.1 *) (* MCP PB 이상리셋 *)
    MCP_SPB_램프_테스트 : BOOL; (* AT %MW87631.2 *) (* MCP SPB LAMP 테스트 *)
    MCP_SPB_부저_정지 : BOOL; (* AT %MW87631.3 *) (* MCP SPB 부저정지 *)
    MCP_TL_GREEN_LAMP : BOOL; (* AT %MW97633.6 *) (* MCP 타워램프 (녹색) *)
    MCP_스피커_멜로디1 : BOOL; (* AT %MW97633.8 *) (* MCP 스피커 멜로디1 (자동기동) *)
    MCP_스피커_멜로디2 : BOOL; (* AT %MW97633.9 *) (* MCP 스피커 멜로디2 (주행) *)
    MCP_스피커_멜로디3 : BOOL; (* AT %MW97633.10 *) (* MCP 스피커 멜로디3 (이상) *)
    MCP_스피커_멜로디4 : BOOL; (* AT %MW97633.11 *) (* MCP 스피커 멜로디4 (경고) *)
    MCP_스피커_멜로디5 : BOOL; (* AT %MW97633.12 *) (* MCP 스피커 멜로디5 (SPARE) *)
    MCP_운전준비_MC_ON : BOOL; (* AT %MW97636.0 *) (* MCP 운전준비 MC ON *)
    MCP_타워_노랑_LAMP : BOOL; (* AT %MW97633.5 *) (* MCP 타워램프 (황색) *)
    MCP_타워_부저 : BOOL; (* AT %MW97633.7 *) (* MCP 타워램프 (부저) *)
    MCP_타워_빨강_LAMP : BOOL; (* AT %MW97633.4 *) (* MCP 타워램프 (적색) *)
END_VAR
VAR
    INST : TON;
    TON_부저_정지 : TON;
    시운전모드 : BOOL;
END_VAR

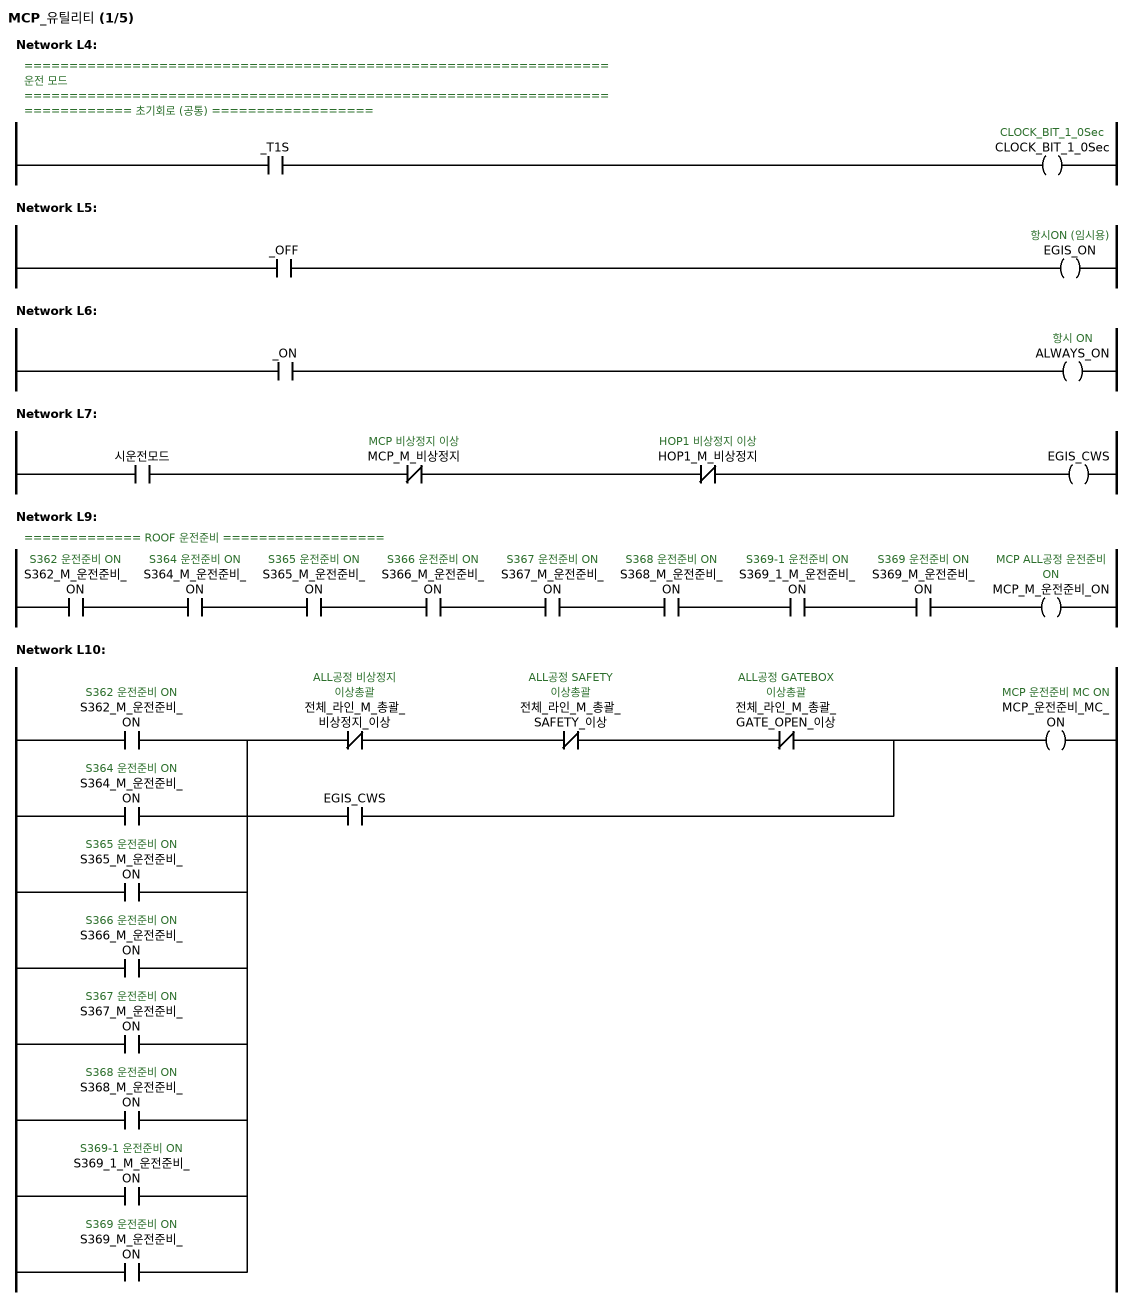
(* ================================================================= *)
(* 운전 모드 *)
(* ================================================================= *)
(* ============ 초기회로 (공통) ================== *)
(* Rung L4 *)
CLOCK_BIT_1_0Sec := _T1S;
(* Rung L5 *)
EGIS_ON := _OFF;
(* Rung L6 *)
ALWAYS_ON := _ON;
(* Rung L7 *)
EGIS_CWS := 시운전모드 AND NOT MCP_M_비상정지 AND NOT HOP1_M_비상정지;
(* ============= ROOF 운전준비 ================== *)
(* Rung L9 *)
MCP_M_운전준비_ON := S362_M_운전준비_ON AND S364_M_운전준비_ON AND S365_M_운전준비_ON AND S366_M_운전준비_ON AND S367_M_운전준비_ON AND S368_M_운전준비_ON AND S369_1_M_운전준비_ON AND S369_M_운전준비_ON;
(* Rung L10 *)
MCP_운전준비_MC_ON := (S362_M_운전준비_ON OR S364_M_운전준비_ON OR S365_M_운전준비_ON OR S366_M_운전준비_ON OR S367_M_운전준비_ON OR S368_M_운전준비_ON OR S369_1_M_운전준비_ON OR S369_M_운전준비_ON) AND ((NOT 전체_라인_M_총괄_비상정지_이상 AND NOT 전체_라인_M_총괄_SAFETY_이상 AND NOT 전체_라인_M_총괄_GATE_OPEN_이상) OR EGIS_CWS);

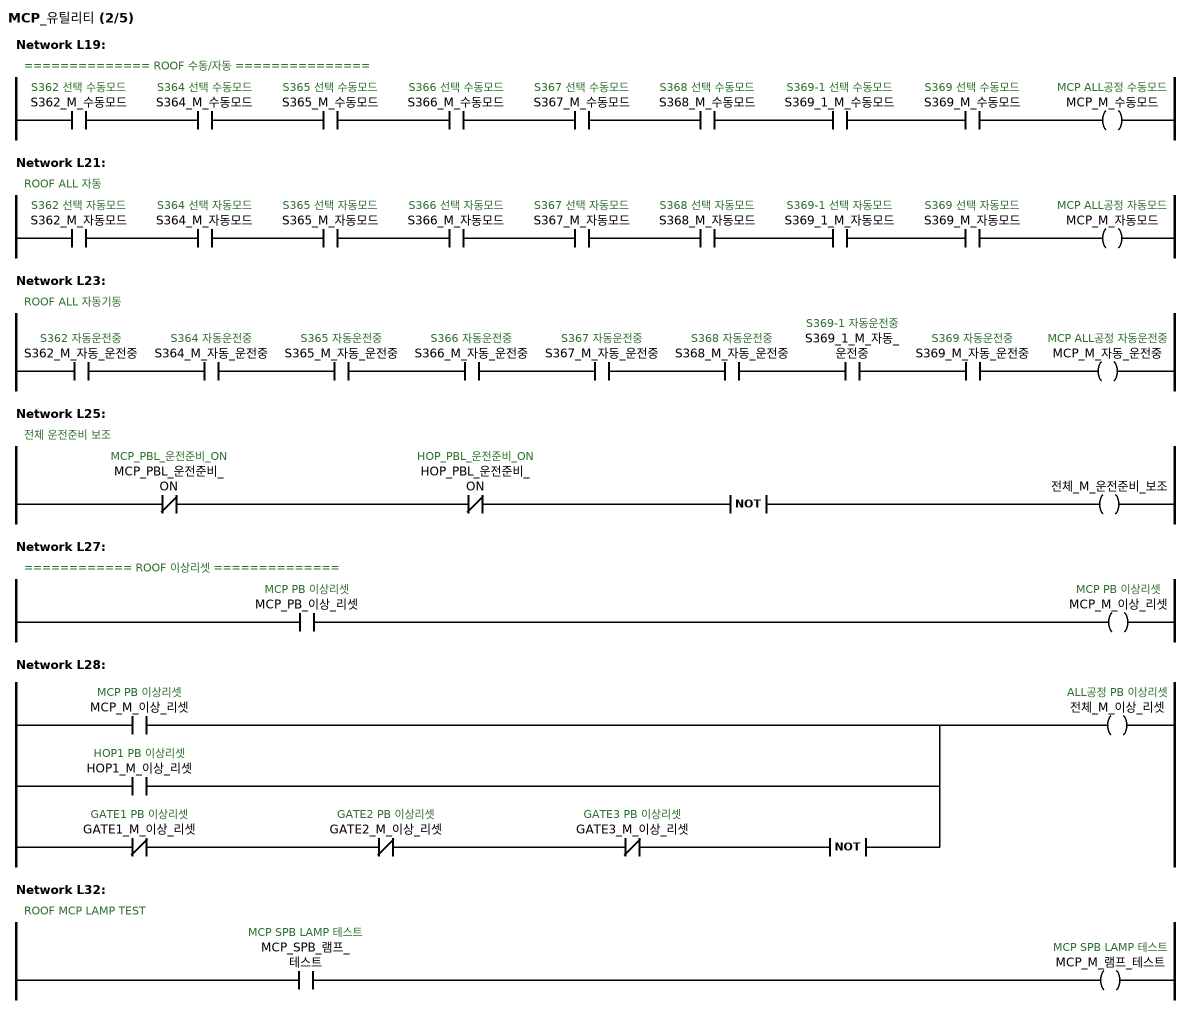
(* ============== ROOF 수동/자동 =============== *)
(* Rung L19 *)
MCP_M_수동모드 := S362_M_수동모드 AND S364_M_수동모드 AND S365_M_수동모드 AND S366_M_수동모드 AND S367_M_수동모드 AND S368_M_수동모드 AND S369_1_M_수동모드 AND S369_M_수동모드;
(* ROOF ALL 자동 *)
(* Rung L21 *)
MCP_M_자동모드 := S362_M_자동모드 AND S364_M_자동모드 AND S365_M_자동모드 AND S366_M_자동모드 AND S367_M_자동모드 AND S368_M_자동모드 AND S369_1_M_자동모드 AND S369_M_자동모드;
(* ROOF ALL 자동기동 *)
(* Rung L23 *)
MCP_M_자동_운전중 := S362_M_자동_운전중 AND S364_M_자동_운전중 AND S365_M_자동_운전중 AND S366_M_자동_운전중 AND S367_M_자동_운전중 AND S368_M_자동_운전중 AND S369_1_M_자동_운전중 AND S369_M_자동_운전중;
(* 전체 운전준비 보조 *)
(* Rung L25 *)
전체_M_운전준비_보조 := NOT (NOT MCP_PBL_운전준비_ON AND NOT HOP_PBL_운전준비_ON);
(* ============ ROOF 이상리셋 ============== *)
(* Rung L27 *)
MCP_M_이상_리셋 := MCP_PB_이상_리셋;
(* Rung L28 *)
전체_M_이상_리셋 := MCP_M_이상_리셋 OR HOP1_M_이상_리셋 OR NOT (NOT GATE1_M_이상_리셋 AND NOT GATE2_M_이상_리셋 AND NOT GATE3_M_이상_리셋);
(* ROOF MCP LAMP TEST *)
(* Rung L32 *)
MCP_M_램프_테스트 := MCP_SPB_램프_테스트;

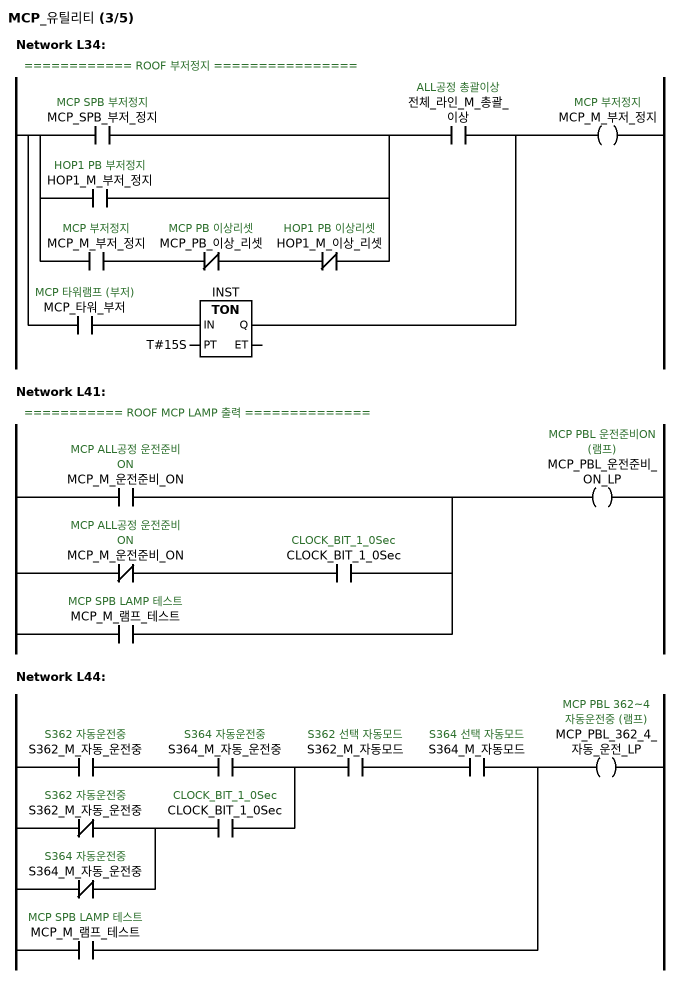
(* ============ ROOF 부저정지 ================ *)
(* Rung L34 *)
INST(IN := MCP_타워_부저, PT := T#15S);
MCP_M_부저_정지 := ((MCP_SPB_부저_정지 OR HOP1_M_부저_정지 OR (MCP_M_부저_정지 AND NOT MCP_PB_이상_리셋 AND NOT HOP1_M_이상_리셋)) AND 전체_라인_M_총괄_이상) OR INST.Q;
(* =========== ROOF MCP LAMP 출력 ============== *)
(* Rung L41 *)
MCP_PBL_운전준비_ON_LP := MCP_M_운전준비_ON OR (NOT MCP_M_운전준비_ON AND CLOCK_BIT_1_0Sec) OR MCP_M_램프_테스트;
(* Rung L44 *)
MCP_PBL_362_4_자동_운전_LP := (((S362_M_자동_운전중 AND S364_M_자동_운전중) OR ((NOT S362_M_자동_운전중 OR NOT S364_M_자동_운전중) AND CLOCK_BIT_1_0Sec)) AND S362_M_자동모드 AND S364_M_자동모드) OR MCP_M_램프_테스트;

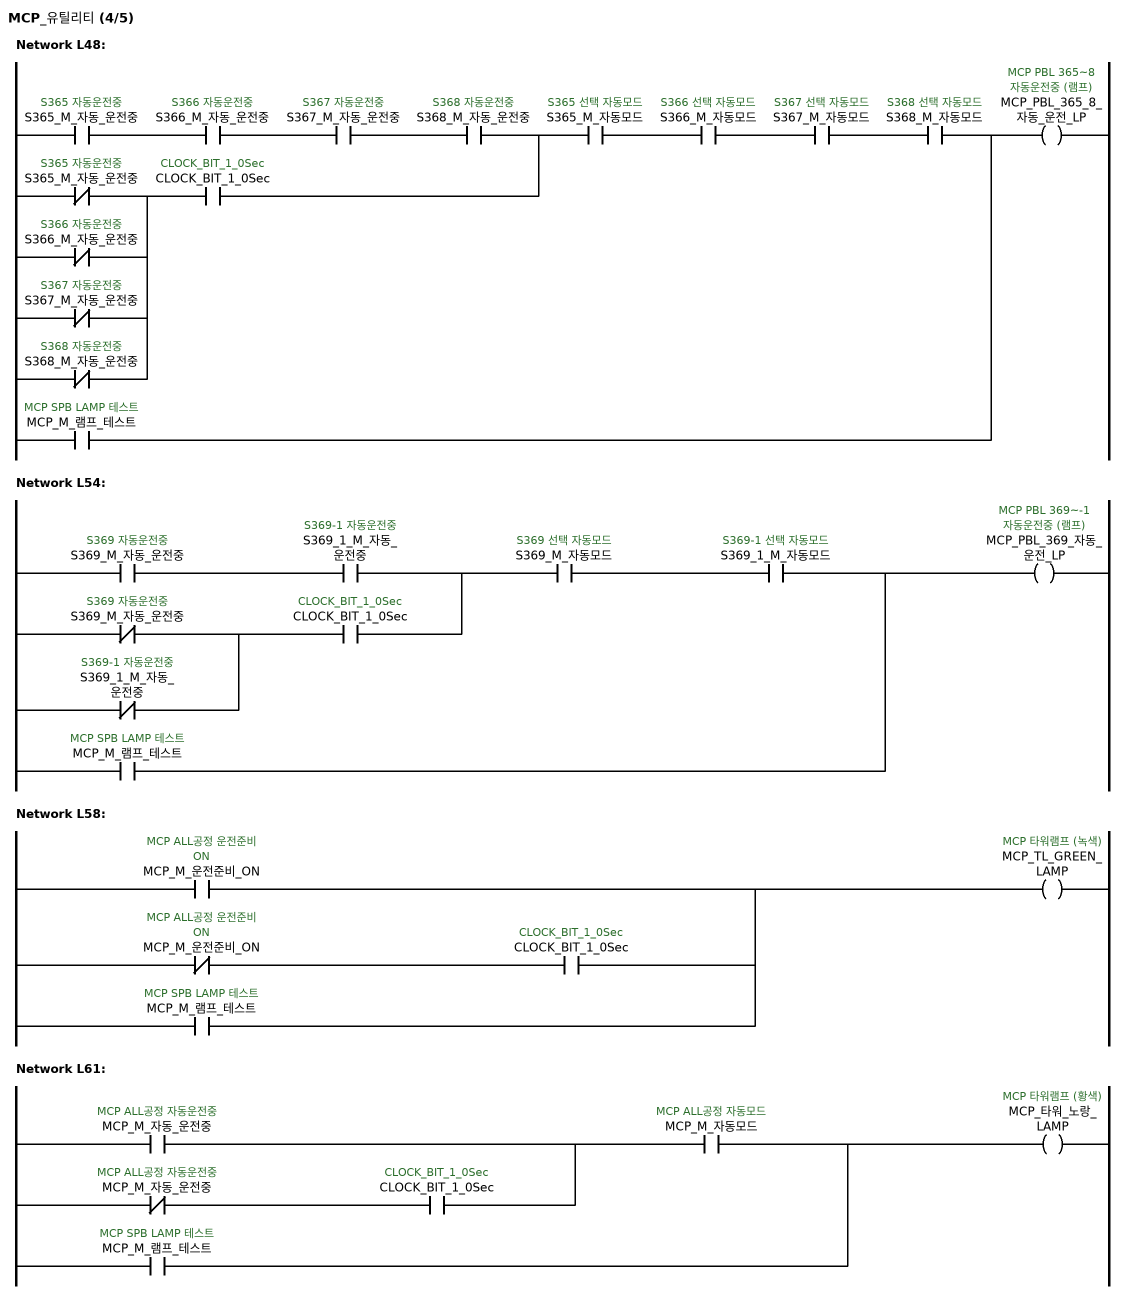
(* Rung L48 *)
MCP_PBL_365_8_자동_운전_LP := (((S365_M_자동_운전중 AND S366_M_자동_운전중 AND S367_M_자동_운전중 AND S368_M_자동_운전중) OR ((NOT S365_M_자동_운전중 OR NOT S366_M_자동_운전중 OR NOT S367_M_자동_운전중 OR NOT S368_M_자동_운전중) AND CLOCK_BIT_1_0Sec)) AND S365_M_자동모드 AND S366_M_자동모드 AND S367_M_자동모드 AND S368_M_자동모드) OR MCP_M_램프_테스트;
(* Rung L54 *)
MCP_PBL_369_자동_운전_LP := (((S369_M_자동_운전중 AND S369_1_M_자동_운전중) OR ((NOT S369_M_자동_운전중 OR NOT S369_1_M_자동_운전중) AND CLOCK_BIT_1_0Sec)) AND S369_M_자동모드 AND S369_1_M_자동모드) OR MCP_M_램프_테스트;
(* Rung L58 *)
MCP_TL_GREEN_LAMP := MCP_M_운전준비_ON OR (NOT MCP_M_운전준비_ON AND CLOCK_BIT_1_0Sec) OR MCP_M_램프_테스트;
(* Rung L61 *)
MCP_타워_노랑_LAMP := ((MCP_M_자동_운전중 OR (NOT MCP_M_자동_운전중 AND CLOCK_BIT_1_0Sec)) AND MCP_M_자동모드) OR MCP_M_램프_테스트;

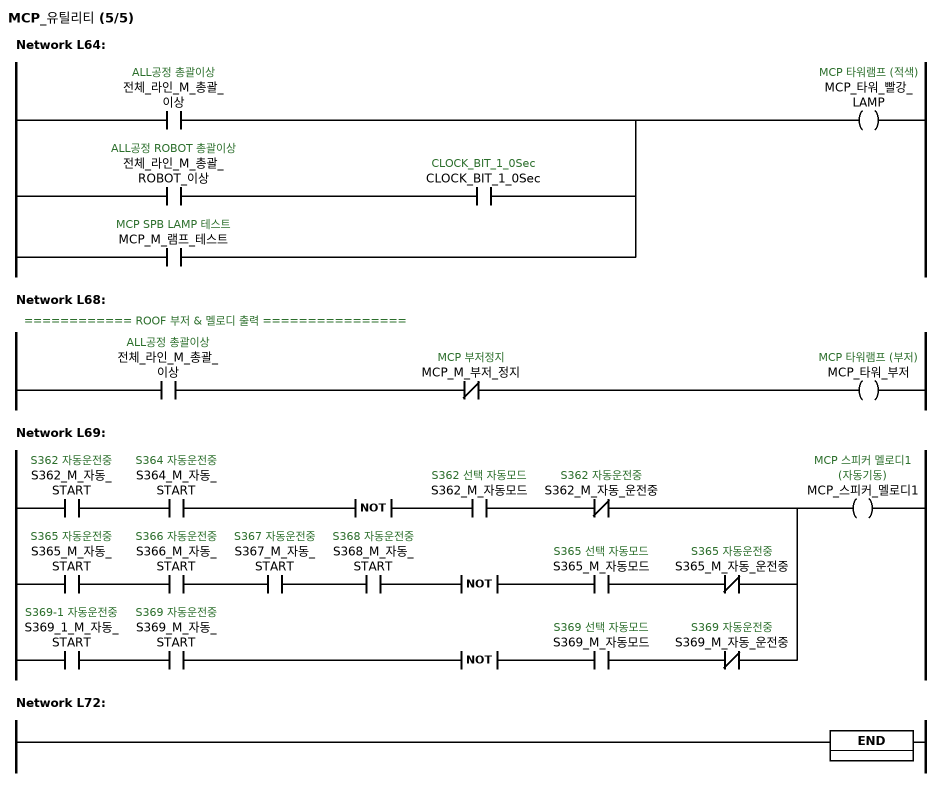
(* Rung L64 *)
MCP_타워_빨강_LAMP := 전체_라인_M_총괄_이상 OR (전체_라인_M_총괄_ROBOT_이상 AND CLOCK_BIT_1_0Sec) OR MCP_M_램프_테스트;
(* ============ ROOF 부저 & 멜로디 출력 ================ *)
(* Rung L68 *)
MCP_타워_부저 := 전체_라인_M_총괄_이상 AND NOT MCP_M_부저_정지;
(* Rung L69 *)
MCP_스피커_멜로디1 := (NOT (S362_M_자동_START AND S364_M_자동_START) AND S362_M_자동모드 AND NOT S362_M_자동_운전중) OR (NOT (S365_M_자동_START AND S366_M_자동_START AND S367_M_자동_START AND S368_M_자동_START) AND S365_M_자동모드 AND NOT S365_M_자동_운전중) OR (NOT (S369_1_M_자동_START AND S369_M_자동_START) AND S369_M_자동모드 AND NOT S369_M_자동_운전중);
(* Rung L72 *)
END();
END_PROGRAM

PROGRAM HOP_유틸리티 (* task: 스캔 프로그램 *)
VAR_EXTERNAL RETAIN
    ALWAYS_OFF : BOOL; (* AT %MW3.0 *) (* 항시 OFF *)
    CLOCK_BIT_1_0Sec : BOOL; (* AT %MW0.5 *) (* CLOCK_BIT_1_0Sec *)
    GATE1_M_CP_TRIP : BOOL; (* AT %MW400.15 *) (* GATEBOX1 CP OFF 이상 *)
    GATE1_M_EMSTOP : BOOL; (* AT %MW400.7 *) (* GATE1 비상정지 이상 *)
    GATE1_M_GATE_CLOSE : BOOL; (* AT %MW400.3 *) (* GATE1_M_GATE_CLOSE *)
    GATE1_M_GATE_열림_보조 : BOOL; (* AT %MW400.12 *) (* GATE1_M_GATE_열림_보조 *)
    GATE1_M_RESTART : BOOL; (* AT %MW400.1 *) (* GATE1_M_RESTART *)
    GATE1_M_STOP_CALL : BOOL; (* AT %MW400.2 *) (* GATE1_M_STOP_CALL *)
    GATE1_M_이상_리셋 : BOOL; (* AT %MW400.0 *) (* GATE1 PB 이상리셋 *)
    GATE1_M_통신_이상 : BOOL; (* AT %MW400.14 *) (* GATEBOX1 통신이상 *)
    GATE2_M_CP_TRIP : BOOL; (* AT %MW401.15 *) (* GATEBOX2 CP OFF 이상 *)
    GATE2_M_EMSTOP : BOOL; (* AT %MW401.7 *) (* GATE2 비상정지 이상 *)
    GATE2_M_GATE_CLOSE : BOOL; (* AT %MW401.3 *) (* GATE2_M_GATE_CLOSE *)
    GATE2_M_GATE_열림_보조 : BOOL; (* AT %MW401.12 *) (* GATE2_M_GATE_열림_보조 *)
    GATE2_M_RESTART : BOOL; (* AT %MW401.1 *) (* GATE2_M_RESTART *)
    GATE2_M_STOP_CALL : BOOL; (* AT %MW401.2 *) (* GATE2_M_STOP_CALL *)
    GATE2_M_이상_리셋 : BOOL; (* AT %MW401.0 *) (* GATE2 PB 이상리셋 *)
    GATE2_M_통신_이상 : BOOL; (* AT %MW401.14 *) (* GATEBOX2 통신이상 *)
    GATE3_M_CP_TRIP : BOOL; (* AT %MW402.15 *) (* GATEBOX3 CP OFF 이상 *)
    GATE3_M_EMSTOP : BOOL; (* AT %MW402.7 *) (* GATE3 비상정지 이상 *)
    GATE3_M_GATE_CLOSE : BOOL; (* AT %MW402.3 *) (* GATE3_M_GATE_CLOSE *)
    GATE3_M_GATE_열림_보조 : BOOL; (* AT %MW402.12 *) (* GATE3_M_GATE_열림_보조 *)
    GATE3_M_RESTART : BOOL; (* AT %MW402.1 *) (* GATE3_M_RESTART *)
    GATE3_M_STOP_CALL : BOOL; (* AT %MW402.2 *) (* GATE3_M_STOP_CALL *)
    GATE3_M_이상_리셋 : BOOL; (* AT %MW402.0 *) (* GATE3 PB 이상리셋 *)
    GATE3_M_통신_이상 : BOOL; (* AT %MW402.14 *) (* GATEBOX3 통신이상 *)
    GATE4_M_CP_TRIP : BOOL; (* AT %MW403.15 *)
    GATE4_M_EMSTOP : BOOL; (* AT %MW403.7 *)
    GATE4_M_GATE_CLOSE : BOOL; (* AT %MW403.3 *)
    GATE4_M_GATE_열림_보조 : BOOL; (* AT %MW403.12 *)
    GATE4_M_RESTART : BOOL; (* AT %MW403.1 *)
    GATE4_M_STOP_CALL : BOOL; (* AT %MW403.2 *)
    GATE4_M_이상_리셋 : BOOL; (* AT %MW403.0 *)
    GATE4_M_통신_이상 : BOOL; (* AT %MW403.14 *)
    GATE5_M_CP_TRIP : BOOL; (* AT %MW404.15 *)
    GATE5_M_EMSTOP : BOOL; (* AT %MW404.7 *)
    GATE5_M_GATE_CLOSE : BOOL; (* AT %MW404.3 *)
    GATE5_M_GATE_열림_보조 : BOOL; (* AT %MW404.12 *)
    GATE5_M_RESTART : BOOL; (* AT %MW404.1 *)
    GATE5_M_STOP_CALL : BOOL; (* AT %MW404.2 *)
    GATE5_M_이상_리셋 : BOOL; (* AT %MW404.0 *)
    GATE5_M_통신_이상 : BOOL; (* AT %MW404.14 *)
    HOP1_M_램프_테스트 : BOOL; (* AT %MW360.6 *) (* HOP1_M_램프_테스트 *)
    HOP1_M_부저_정지 : BOOL; (* AT %MW360.5 *) (* HOP1 PB 부저정지 *)
    HOP1_M_수동모드 : BOOL; (* AT %MW360.1 *) (* HOP1_M_수동모드 *)
    HOP1_M_운전준비_ON : BOOL; (* AT %MW360.0 *) (* HOP1_M_운전준비_ON *)
    HOP1_M_이상_리셋 : BOOL; (* AT %MW360.4 *) (* HOP1 PB 이상리셋 *)
    HOP1_M_자동_START : BOOL; (* AT %MW360.3 *) (* HOP1_M_자동_START *)
    MCP_M_운전준비_ON : BOOL; (* AT %MW350.0 *) (* MCP ALL공정 운전준비 ON *)
    MCP_M_이상_리셋 : BOOL; (* AT %MW350.4 *) (* MCP PB 이상리셋 *)
    MCP_M_자동_운전중 : BOOL; (* AT %MW350.3 *) (* MCP ALL공정 자동운전중 *)
    MCP_M_자동모드 : BOOL; (* AT %MW350.2 *) (* MCP ALL공정 자동모드 *)
    S362_M_자동_운전중 : BOOL; (* AT %MW1000.4 *) (* S362 자동운전중 *)
    S364_M_자동_운전중 : BOOL; (* AT %MW2000.4 *) (* S364 자동운전중 *)
    S365_M_자동_운전중 : BOOL; (* AT %MW2500.4 *) (* S365 자동운전중 *)
    S366_M_자동_운전중 : BOOL; (* AT %MW3000.4 *) (* S366 자동운전중 *)
    S367_M_자동_운전중 : BOOL; (* AT %MW3500.4 *) (* S367 자동운전중 *)
    S368_M_자동_운전중 : BOOL; (* AT %MW4000.4 *) (* S368 자동운전중 *)
    S369_1_M_자동_운전중 : BOOL; (* AT %MW4500.4 *) (* S369-1 자동운전중 *)
    S369_M_자동_운전중 : BOOL; (* AT %MW5000.4 *) (* S369 자동운전중 *)
    전체_M_CYCLE_정지 : BOOL; (* AT %MW308.0 *) (* 전체_M_CYCLE_정지 *)
    전체_M_GATE_자동기동 : BOOL; (* AT %MW308.1 *) (* 전체_M_자동_운전 *)
    전체_M_OPEN_조건 : BOOL; (* AT %MW308.3 *) (* 전체_M_OPEN_조건 *)
    전체_M_이상_리셋 : BOOL; (* AT %MW308.2 *) (* ALL공정 PB 이상리셋 *)
    전체_라인_M_총괄_이상 : BOOL; (* AT %MW300.0 *) (* ALL공정 총괄이상 *)
END_VAR
VAR_EXTERNAL
    GB1_7_1_PLC_BOX_CP_TRIP : BOOL; (* AT %MW87010.15 *) (* GB1_7_1_PLC_BOX_CP_TRIP *)
    GB1_PBL_CYCLE_정지 : BOOL; (* AT %MW87010.1 *) (* GB1_PBL_CYCLE_정지 *)
    GB1_PBL_CYCLE_정지_LAMP : BOOL; (* AT %MW97011.1 *) (* GB1_PBL_CYCLE_정지_LAMP *)
    GB1_PBL_자동_운전 : BOOL; (* AT %MW87010.0 *) (* GB1_PBL_자동_운전 *)
    GB1_PBL_자동_운전_LAMP : BOOL; (* AT %MW97011.0 *) (* GB1_PBL_자동_운전_LAMP *)
    GB1_PB_이상_리셋 : BOOL; (* AT %MW87010.2 *) (* GB1_PB_이상_리셋 *)
    GB1_SAFETY_DOOR_LOCK1 : BOOL; (* AT %MW87012.8 *)
    GB1_SAFETY_DOOR_LOOK2 : BOOL; (* AT %MW87012.9 *)
    GB1_SAFETY_DOOR_UNLOOK1 : BOOL; (* AT %MW97013.0 *) (* GB1_SAFETY_DOOR_UNLOOK1 *)
    GB1_SAFETY_DOOR_UNLOOK2 : BOOL; (* AT %MW97013.1 *) (* GB1_SAFETY_DOOR_UNLOOK2 *)
    GB1_TL_GREEN_LAMP : BOOL; (* AT %MW97011.9 *) (* GB1_TL_GREEN_LAMP *)
    GB1_TL_RED_LAMP : BOOL; (* AT %MW97011.8 *) (* GB1_TL_RED_LAMP *)
    GB2_7_2_PLC_BOX_CP_TRIP : BOOL; (* AT %MW87020.15 *) (* GB2_7_2_PLC_BOX_CP_TRIP *)
    GB2_PBL_CYCLE_정지 : BOOL; (* AT %MW87020.1 *) (* GB2_PBL_CYCLE_정지 *)
    GB2_PBL_CYCLE_정지_LAMP : BOOL; (* AT %MW97021.1 *) (* GB2_PBL_CYCLE_정지_LAMP *)
    GB2_PBL_자동_운전 : BOOL; (* AT %MW87020.0 *) (* GB2_PBL_자동_운전 *)
    GB2_PBL_자동_운전_LAMP : BOOL; (* AT %MW97021.0 *) (* GB2_PBL_자동_운전_LAMP *)
    GB2_PB_이상_리셋 : BOOL; (* AT %MW87020.2 *) (* GB2_PB_이상_리셋 *)
    GB2_SAFETY_DOOR_LOCK1 : BOOL; (* AT %MW87022.8 *) (* GB2_SAFETY_DOOR_LOCK1 *)
    GB2_SAFETY_DOOR_LOOK2 : BOOL; (* AT %MW87022.9 *) (* GB2_SAFETY_DOOR_LOOK2 *)
    GB2_SAFETY_DOOR_UNLOOK1 : BOOL; (* AT %MW97023.0 *) (* GB2_SAFETY_DOOR_UNLOOK1 *)
    GB2_SAFETY_DOOR_UNLOOK2 : BOOL; (* AT %MW97023.1 *) (* GB2_SAFETY_DOOR_UNLOOK2 *)
    GB2_TL_GREEN_LAMP : BOOL; (* AT %MW97021.9 *) (* GB2_TL_GREEN_LAMP *)
    GB2_TL_RED_LAMP : BOOL; (* AT %MW97021.8 *) (* GB2_TL_RED_LAMP *)
    GB3_7_3_PLC_BOX_CP_TRIP : BOOL; (* AT %MW87030.15 *) (* GB3_7_3_PLC_BOX_CP_TRIP *)
    GB3_PBL_CYCLE_정지 : BOOL; (* AT %MW87030.1 *) (* GB3_PBL_CYCLE_정지 *)
    GB3_PBL_CYCLE_정지_LAMP : BOOL; (* AT %MW97031.1 *) (* GB3_PBL_CYCLE_정지_LAMP *)
    GB3_PBL_자동_운전 : BOOL; (* AT %MW87030.0 *) (* GB3_PBL_자동_운전 *)
    GB3_PBL_자동_운전_LAMP : BOOL; (* AT %MW97031.0 *) (* GB3_PBL_자동_운전_LAMP *)
    GB3_PB_이상_리셋 : BOOL; (* AT %MW87030.2 *) (* GB3_PB_이상_리셋 *)
    GB3_SAFETY_DOOR_LOCK1 : BOOL; (* AT %MW87032.8 *) (* GB3_SAFETY_DOOR_LOCK1 *)
    GB3_SAFETY_DOOR_LOOK2 : BOOL; (* AT %MW87032.9 *) (* GB3_SAFETY_DOOR_LOOK2 *)
    GB3_SAFETY_DOOR_UNLOOK1 : BOOL; (* AT %MW97033.0 *) (* GB3_SAFETY_DOOR_UNLOOK1 *)
    GB3_SAFETY_DOOR_UNLOOK2 : BOOL; (* AT %MW97033.1 *) (* GB3_SAFETY_DOOR_UNLOOK2 *)
    GB3_TL_GREEN_LAMP : BOOL; (* AT %MW97031.9 *) (* GB3_TL_GREEN_LAMP *)
    GB3_TL_RED_LAMP : BOOL; (* AT %MW97031.8 *) (* GB3_TL_RED_LAMP *)
    GB4_7_11_PLC_BOX_CP_TRIP : BOOL; (* AT %MW87110.15 *) (* GB4 7 11 PLC BOX CP TRIP *)
    GB4_7_3_PLC_BOX_CP_TRIP : BOOL; (* GB3_7_3_PLC_BOX_CP_TRIP *)
    GB4_PBL_CYCLE_정지 : BOOL; (* AT %MW87110.1 *) (* GB4 PBL CYCLE 정지 *)
    GB4_PBL_CYCLE_정지_LAMP : BOOL; (* AT %MW97111.1 *) (* GB4 PBL CYCLE 정지 LAMP *)
    GB4_PBL_자동_운전 : BOOL; (* AT %MW87110.0 *) (* GB4 PBL 자동 운전 *)
    GB4_PBL_자동_운전_LAMP : BOOL; (* AT %MW97111.0 *) (* GB4 PBL 자동 운전 LAMP *)
    GB4_PB_이상_리셋 : BOOL; (* AT %MW87110.2 *) (* GB4 PB 이상 리셋 *)
    GB4_SAFETY_DOOR_LOCK1 : BOOL; (* AT %MW87112.8 *) (* GB4 SAFETY DOOR LOCK1 *)
    GB4_SAFETY_DOOR_LOOK2 : BOOL; (* AT %MW87112.9 *) (* GB4 SAFETY DOOR LOCK2 *)
    GB4_SAFETY_DOOR_UNLOOK1 : BOOL; (* AT %MW97113.0 *) (* GB4 SAFETY DOOR UNLOOK1 *)
    GB4_SAFETY_DOOR_UNLOOK2 : BOOL; (* AT %MW97113.1 *) (* GB4 SAFETY DOOR UNLOOK2 *)
    GB4_TL_GREEN_LAMP : BOOL; (* AT %MW97111.9 *) (* GB4 TL GREEN LAMP *)
    GB4_TL_RED_LAMP : BOOL; (* AT %MW97111.8 *) (* GB4 TL RED LAMP *)
    GB5_7_11_PLC_BOX_CP_TRIP : BOOL; (* GB4 7 11 PLC BOX CP TRIP *)
    GB5_7_12_PLC_BOX_CP_TRIP : BOOL; (* AT %MW87120.15 *) (* GB5 7 12 PLC BOX CP TRIP *)
    GB5_PBL_CYCLE_정지 : BOOL; (* AT %MW87120.1 *) (* GB5 PBL CYCLE 정지 *)
    GB5_PBL_CYCLE_정지_LAMP : BOOL; (* AT %MW97121.1 *) (* GB5 PBL CYCLE 정지 LAMP *)
    GB5_PBL_자동_운전 : BOOL; (* AT %MW87120.0 *) (* GB5 PBL 자동 운전 *)
    GB5_PBL_자동_운전_LAMP : BOOL; (* AT %MW97121.0 *) (* GB5 PBL 자동 운전 LAMP *)
    GB5_PB_이상_리셋 : BOOL; (* AT %MW87120.2 *) (* GB5 PB 이상 리셋 *)
    GB5_SAFETY_DOOR_LOCK1 : BOOL; (* AT %MW87122.8 *) (* GB5 SAFETY DOOR LOCK1 *)
    GB5_SAFETY_DOOR_LOOK2 : BOOL; (* AT %MW87122.9 *) (* GB5 SAFETY DOOR LOCK2 *)
    GB5_SAFETY_DOOR_UNLOOK1 : BOOL; (* AT %MW97123.0 *) (* GB5 SAFETY DOOR UNLOOK1 *)
    GB5_SAFETY_DOOR_UNLOOK2 : BOOL; (* AT %MW97123.1 *) (* GB5 SAFETY DOOR UNLOOK2 *)
    GB5_TL_GREEN_LAMP : BOOL; (* AT %MW97121.9 *) (* GB5 TL GREEN LAMP *)
    GB5_TL_RED_LAMP : BOOL; (* AT %MW97121.8 *) (* GB5 TL RED LAMP *)
    HOP_PBL_362_4_자동_운전_LP : BOOL; (* AT %MW97502.1 *) (* HOP_PBL_362_4_자동_운전_LP *)
    HOP_PBL_365_8_자동_운전_LP : BOOL; (* AT %MW97502.2 *) (* HOP_PBL_365_8_자동_운전_LP *)
    HOP_PBL_369_자동_운전_LP : BOOL; (* AT %MW97502.3 *) (* HOP_PBL_369_자동_운전_LP *)
    HOP_PBL_운전준비_ON : BOOL; (* AT %MW87500.0 *) (* HOP_PBL_운전준비_ON *)
    HOP_PBL_운전준비_ON_LP : BOOL; (* AT %MW97502.0 *) (* HOP_PBL_운전준비_ON_LP *)
    HOP_PB_이상_리셋 : BOOL; (* AT %MW87500.1 *) (* HOP_PB_이상_리셋 *)
    HOP_SPB_램프_테스트 : BOOL; (* AT %MW87500.11 *) (* HOP_SPB_램프_테스트 *)
    HOP_SPB_부저_정지 : BOOL; (* AT %MW87500.12 *) (* HOP_SPB_부저_정지 *)
    HOP_부저 : BOOL; (* AT %MW97502.10 *) (* HOP_부저 *)
    HOP_타워_빨강_LP : BOOL; (* AT %MW97502.7 *) (* HOP_타워_빨강_LP *)
    MCP_타워_부저 : BOOL; (* AT %MW97633.7 *) (* MCP 타워램프 (부저) *)
    _0007_EB01_CFG_ER : BOOL; (* AT %MW187022.0 *) (* EB 구성 에러 *)
    _0007_EB01_DEER : BOOL; (* AT %MW187022.1 *) (* EB 운전 중 탈락 *)
    _0007_EB01_IO_DEER : BOOL; (* AT %MW187023.2 *) (* EB IO 탈락 에러 *)
    _0007_EB01_IO_TYER : BOOL; (* AT %MW187023.1 *) (* EB IO 타입 에러 *)
    _0007_EB02_CFG_ER : BOOL; (* AT %MW187028.0 *) (* EB 구성 에러 *)
    _0007_EB02_DEER : BOOL; (* AT %MW187028.1 *) (* EB 운전 중 탈락 *)
    _0007_EB02_IO_DEER : BOOL; (* AT %MW187029.2 *) (* EB IO 탈락 에러 *)
    _0007_EB02_IO_TYER : BOOL; (* AT %MW187029.1 *) (* EB IO 타입 에러 *)
    _0007_EB03_CFG_ER : BOOL; (* AT %MW187034.0 *) (* EB 구성 에러 *)
    _0007_EB03_DEER : BOOL; (* AT %MW187034.1 *) (* EB 운전 중 탈락 *)
    _0007_EB03_IO_DEER : BOOL; (* AT %MW187035.2 *) (* EB IO 탈락 에러 *)
    _0007_EB03_IO_TYER : BOOL; (* AT %MW187035.1 *) (* EB IO 타입 에러 *)
    _0007_EB11_CFG_ER : BOOL; (* AT %MW187046.0 *) (* EB 구성 에러 *)
    _0007_EB11_DEER : BOOL; (* AT %MW187046.1 *) (* EB 운전 중 탈락 *)
    _0007_EB11_IO_DEER : BOOL; (* AT %MW187047.2 *) (* EB IO 탈락 에러 *)
    _0007_EB11_IO_TYER : BOOL; (* AT %MW187047.1 *) (* EB IO 타입 에러 *)
    _0007_EB12_CFG_ER : BOOL; (* AT %MW187052.0 *) (* EB 구성 에러 *)
    _0007_EB12_DEER : BOOL; (* AT %MW187052.1 *) (* EB 운전 중 탈락 *)
    _0007_EB12_IO_DEER : BOOL; (* AT %MW187053.2 *) (* EB IO 탈락 에러 *)
    _0007_EB12_IO_TYER : BOOL; (* AT %MW187053.1 *) (* EB IO 타입 에러 *)
    _0007_EB40_CFG_ER : BOOL; (* AT %MW187070.0 *) (* EB 구성 에러 *)
    _0007_EB40_DEER : BOOL; (* AT %MW187070.1 *) (* EB 운전 중 탈락 *)
    _0007_EB40_IO_DEER : BOOL; (* AT %MW187071.2 *) (* EB IO 탈락 에러 *)
    _0007_EB40_IO_TYER : BOOL; (* AT %MW187071.1 *) (* EB IO 타입 에러 *)
END_VAR
VAR
    TON_GATE10_OPEN : TON;
    TON_GATE11_OPEN : TON;
    TON_GATE1_OPEN : TON;
    TON_GATE2_OPEN : TON;
    TON_GATE3_OPEN : TON;
    TON_GATE4_OPEN : TON;
    TON_GATE5_OPEN : TON;
    TON_GATE6_OPEN : TON;
    TON_GATE7_OPEN : TON;
    TON_GATE8_OPEN : TON;
    TON_GATE9_OPEN : TON;
    T_GB1_CP_OFF_DELAY : TON;
    T_GB1_통신_이상_DELAY : TON;
    T_GB2_CP_OFF_DELAY : TON;
    T_GB2_통신_이상_DELAY : TON;
    T_GB3_CP_OFF_DELAY : TON;
    T_GB3_통신_이상_DELAY : TON;
    T_GB4_CP_OFF_DELAY : TON;
    T_GB4_통신_이상_DELAY : TON;
    T_GB5_CP_OFF_DELAY : TON;
    T_GB5_통신_이상_DELAY : TON;
END_VAR

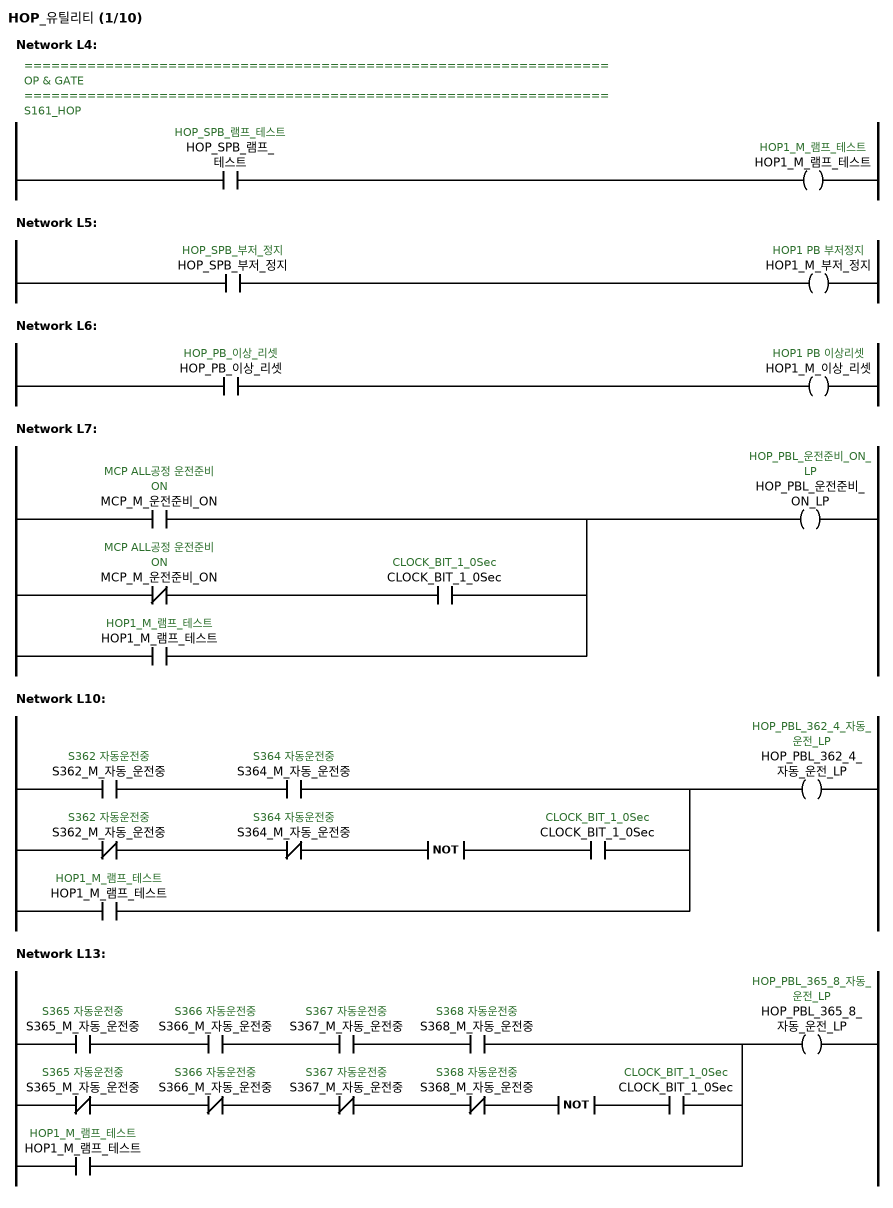
(* ================================================================= *)
(* OP & GATE *)
(* ================================================================= *)
(* S161_HOP *)
(* Rung L4 *)
HOP1_M_램프_테스트 := HOP_SPB_램프_테스트;
(* Rung L5 *)
HOP1_M_부저_정지 := HOP_SPB_부저_정지;
(* Rung L6 *)
HOP1_M_이상_리셋 := HOP_PB_이상_리셋;
(* Rung L7 *)
HOP_PBL_운전준비_ON_LP := MCP_M_운전준비_ON OR (NOT MCP_M_운전준비_ON AND CLOCK_BIT_1_0Sec) OR HOP1_M_램프_테스트;
(* Rung L10 *)
HOP_PBL_362_4_자동_운전_LP := (S362_M_자동_운전중 AND S364_M_자동_운전중) OR (NOT (NOT S362_M_자동_운전중 AND NOT S364_M_자동_운전중) AND CLOCK_BIT_1_0Sec) OR HOP1_M_램프_테스트;
(* Rung L13 *)
HOP_PBL_365_8_자동_운전_LP := (S365_M_자동_운전중 AND S366_M_자동_운전중 AND S367_M_자동_운전중 AND S368_M_자동_운전중) OR (NOT (NOT S365_M_자동_운전중 AND NOT S366_M_자동_운전중 AND NOT S367_M_자동_운전중 AND NOT S368_M_자동_운전중) AND CLOCK_BIT_1_0Sec) OR HOP1_M_램프_테스트;

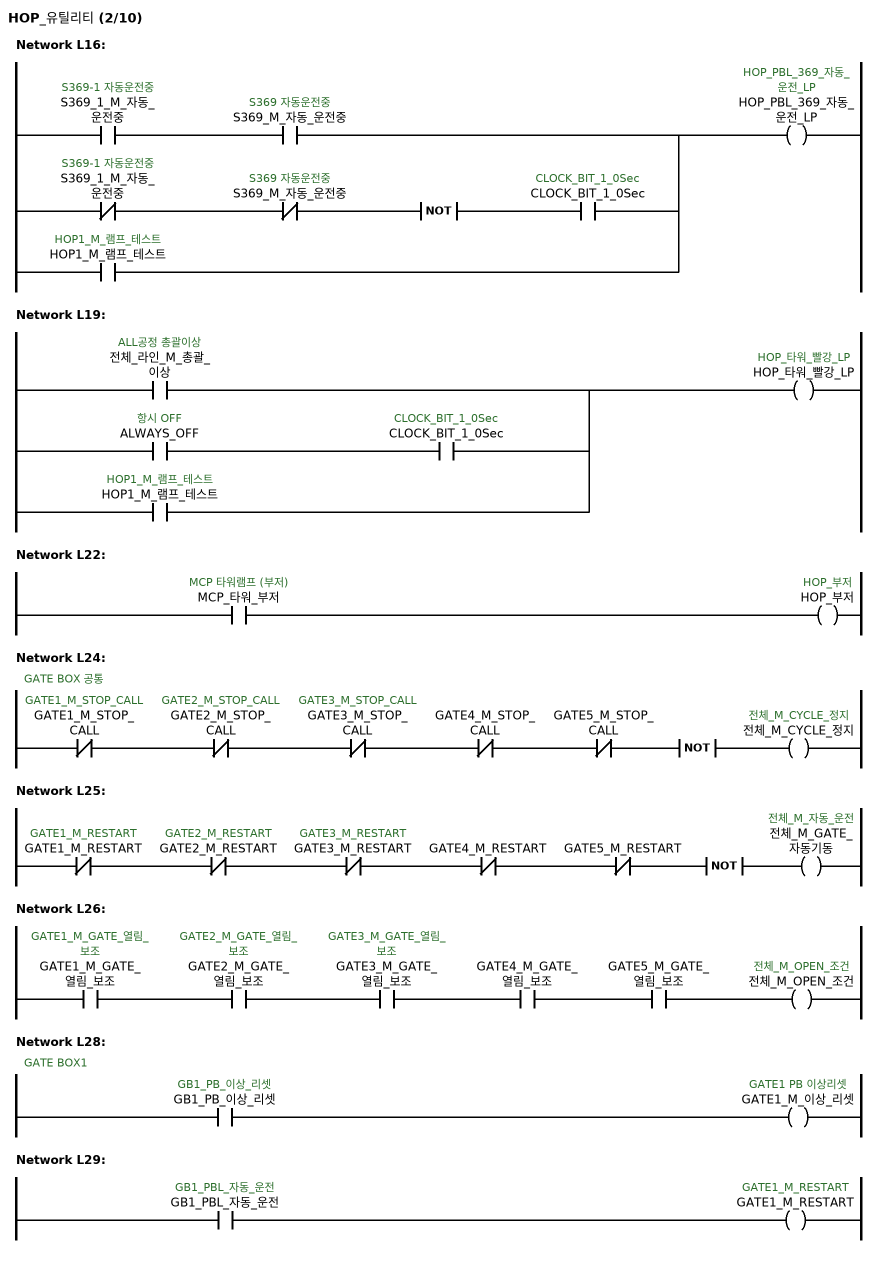
(* Rung L16 *)
HOP_PBL_369_자동_운전_LP := (S369_1_M_자동_운전중 AND S369_M_자동_운전중) OR (NOT (NOT S369_1_M_자동_운전중 AND NOT S369_M_자동_운전중) AND CLOCK_BIT_1_0Sec) OR HOP1_M_램프_테스트;
(* Rung L19 *)
HOP_타워_빨강_LP := 전체_라인_M_총괄_이상 OR (ALWAYS_OFF AND CLOCK_BIT_1_0Sec) OR HOP1_M_램프_테스트;
(* Rung L22 *)
HOP_부저 := MCP_타워_부저;
(* GATE BOX 공통 *)
(* Rung L24 *)
전체_M_CYCLE_정지 := NOT (NOT GATE1_M_STOP_CALL AND NOT GATE2_M_STOP_CALL AND NOT GATE3_M_STOP_CALL AND NOT GATE4_M_STOP_CALL AND NOT GATE5_M_STOP_CALL);
(* Rung L25 *)
전체_M_GATE_자동기동 := NOT (NOT GATE1_M_RESTART AND NOT GATE2_M_RESTART AND NOT GATE3_M_RESTART AND NOT GATE4_M_RESTART AND NOT GATE5_M_RESTART);
(* Rung L26 *)
전체_M_OPEN_조건 := GATE1_M_GATE_열림_보조 AND GATE2_M_GATE_열림_보조 AND GATE3_M_GATE_열림_보조 AND GATE4_M_GATE_열림_보조 AND GATE5_M_GATE_열림_보조;
(* GATE BOX1 *)
(* Rung L28 *)
GATE1_M_이상_리셋 := GB1_PB_이상_리셋;
(* Rung L29 *)
GATE1_M_RESTART := GB1_PBL_자동_운전;

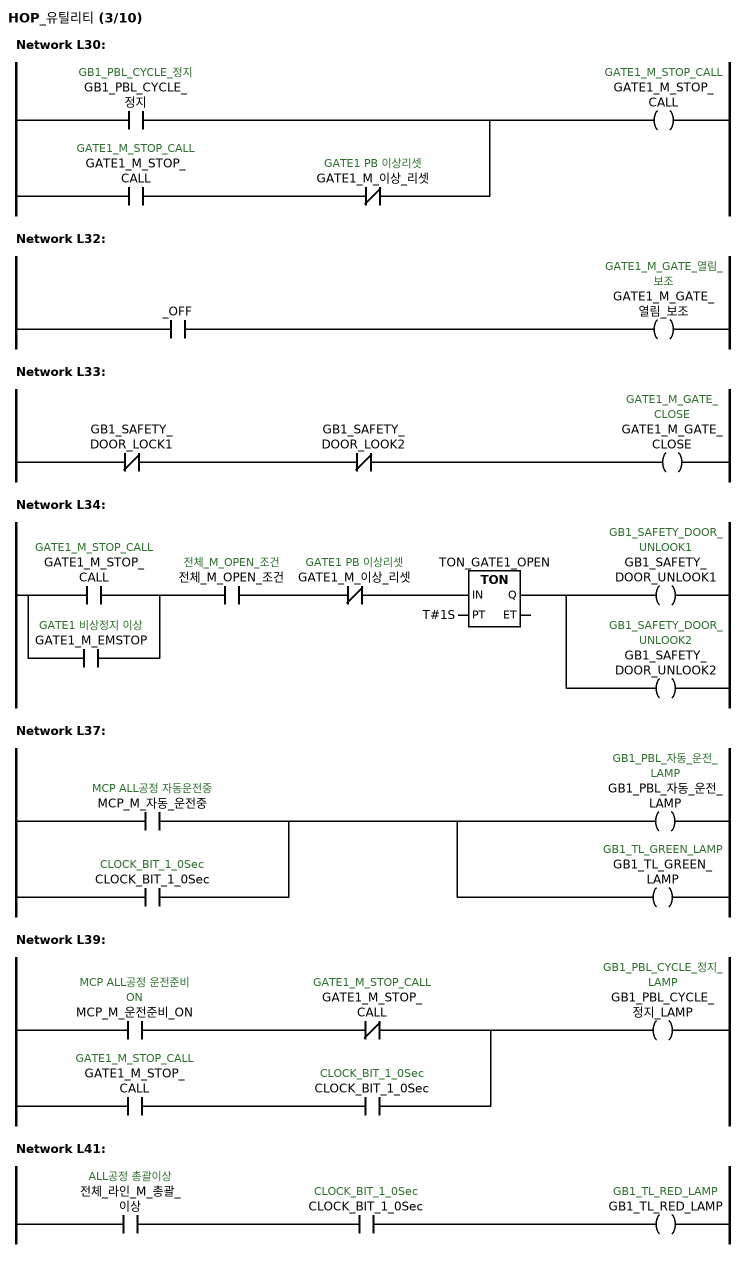
(* Rung L30 *)
GATE1_M_STOP_CALL := GB1_PBL_CYCLE_정지 OR (GATE1_M_STOP_CALL AND NOT GATE1_M_이상_리셋);
(* Rung L32 *)
GATE1_M_GATE_열림_보조 := _OFF;
(* Rung L33 *)
GATE1_M_GATE_CLOSE := NOT GB1_SAFETY_DOOR_LOCK1 AND NOT GB1_SAFETY_DOOR_LOOK2;
(* Rung L34 *)
TON_GATE1_OPEN(IN := (GATE1_M_STOP_CALL OR GATE1_M_EMSTOP) AND 전체_M_OPEN_조건 AND NOT GATE1_M_이상_리셋, PT := T#1S);
GB1_SAFETY_DOOR_UNLOOK1 := TON_GATE1_OPEN.Q;
GB1_SAFETY_DOOR_UNLOOK2 := TON_GATE1_OPEN.Q;
(* Rung L37 *)
GB1_PBL_자동_운전_LAMP := MCP_M_자동_운전중 OR CLOCK_BIT_1_0Sec;
GB1_TL_GREEN_LAMP := MCP_M_자동_운전중 OR CLOCK_BIT_1_0Sec;
(* Rung L39 *)
GB1_PBL_CYCLE_정지_LAMP := (MCP_M_운전준비_ON AND NOT GATE1_M_STOP_CALL) OR (GATE1_M_STOP_CALL AND CLOCK_BIT_1_0Sec);
(* Rung L41 *)
GB1_TL_RED_LAMP := 전체_라인_M_총괄_이상 AND CLOCK_BIT_1_0Sec;

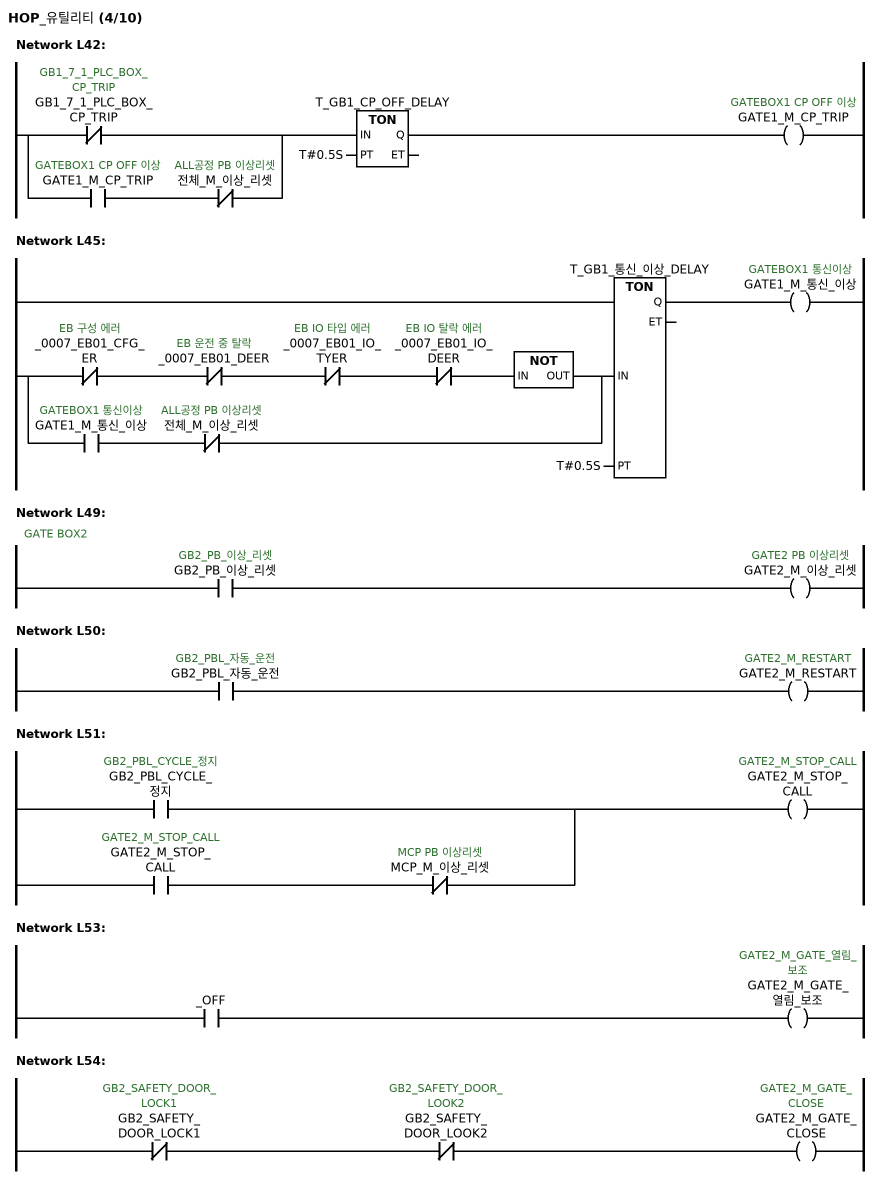
(* Rung L42 *)
T_GB1_CP_OFF_DELAY(IN := NOT GB1_7_1_PLC_BOX_CP_TRIP OR (GATE1_M_CP_TRIP AND NOT 전체_M_이상_리셋), PT := T#0.5S);
GATE1_M_CP_TRIP := T_GB1_CP_OFF_DELAY.Q;
(* Rung L45 *)
T_GB1_통신_이상_DELAY(IN := (NOT (NOT _0007_EB01_CFG_ER AND NOT _0007_EB01_DEER AND NOT _0007_EB01_IO_TYER AND NOT _0007_EB01_IO_DEER)) OR (GATE1_M_통신_이상 AND NOT 전체_M_이상_리셋), PT := T#0.5S);
GATE1_M_통신_이상 := T_GB1_통신_이상_DELAY.Q;
(* GATE BOX2 *)
(* Rung L49 *)
GATE2_M_이상_리셋 := GB2_PB_이상_리셋;
(* Rung L50 *)
GATE2_M_RESTART := GB2_PBL_자동_운전;
(* Rung L51 *)
GATE2_M_STOP_CALL := GB2_PBL_CYCLE_정지 OR (GATE2_M_STOP_CALL AND NOT MCP_M_이상_리셋);
(* Rung L53 *)
GATE2_M_GATE_열림_보조 := _OFF;
(* Rung L54 *)
GATE2_M_GATE_CLOSE := NOT GB2_SAFETY_DOOR_LOCK1 AND NOT GB2_SAFETY_DOOR_LOOK2;

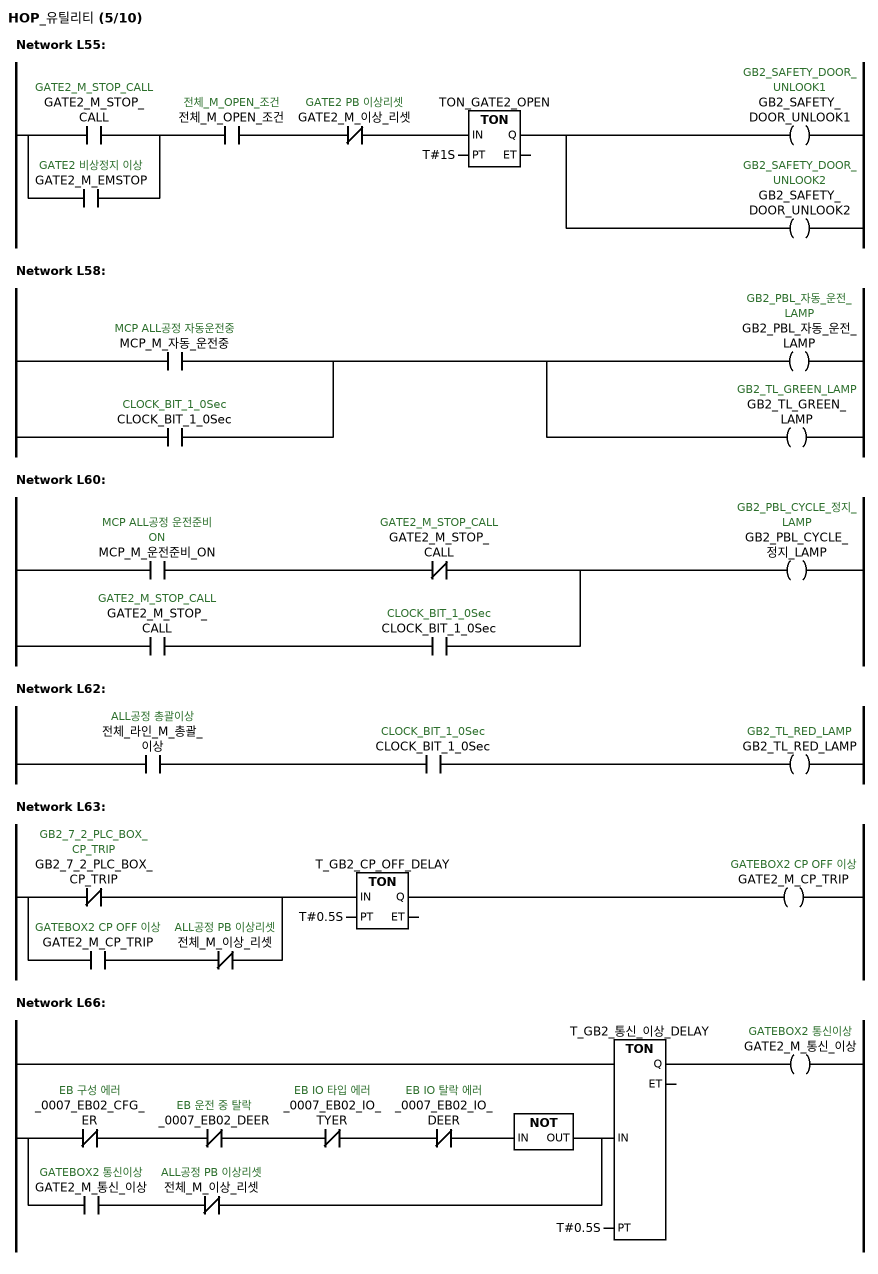
(* Rung L55 *)
TON_GATE2_OPEN(IN := (GATE2_M_STOP_CALL OR GATE2_M_EMSTOP) AND 전체_M_OPEN_조건 AND NOT GATE2_M_이상_리셋, PT := T#1S);
GB2_SAFETY_DOOR_UNLOOK1 := TON_GATE2_OPEN.Q;
GB2_SAFETY_DOOR_UNLOOK2 := TON_GATE2_OPEN.Q;
(* Rung L58 *)
GB2_PBL_자동_운전_LAMP := MCP_M_자동_운전중 OR CLOCK_BIT_1_0Sec;
GB2_TL_GREEN_LAMP := MCP_M_자동_운전중 OR CLOCK_BIT_1_0Sec;
(* Rung L60 *)
GB2_PBL_CYCLE_정지_LAMP := (MCP_M_운전준비_ON AND NOT GATE2_M_STOP_CALL) OR (GATE2_M_STOP_CALL AND CLOCK_BIT_1_0Sec);
(* Rung L62 *)
GB2_TL_RED_LAMP := 전체_라인_M_총괄_이상 AND CLOCK_BIT_1_0Sec;
(* Rung L63 *)
T_GB2_CP_OFF_DELAY(IN := NOT GB2_7_2_PLC_BOX_CP_TRIP OR (GATE2_M_CP_TRIP AND NOT 전체_M_이상_리셋), PT := T#0.5S);
GATE2_M_CP_TRIP := T_GB2_CP_OFF_DELAY.Q;
(* Rung L66 *)
T_GB2_통신_이상_DELAY(IN := (NOT (NOT _0007_EB02_CFG_ER AND NOT _0007_EB02_DEER AND NOT _0007_EB02_IO_TYER AND NOT _0007_EB02_IO_DEER)) OR (GATE2_M_통신_이상 AND NOT 전체_M_이상_리셋), PT := T#0.5S);
GATE2_M_통신_이상 := T_GB2_통신_이상_DELAY.Q;

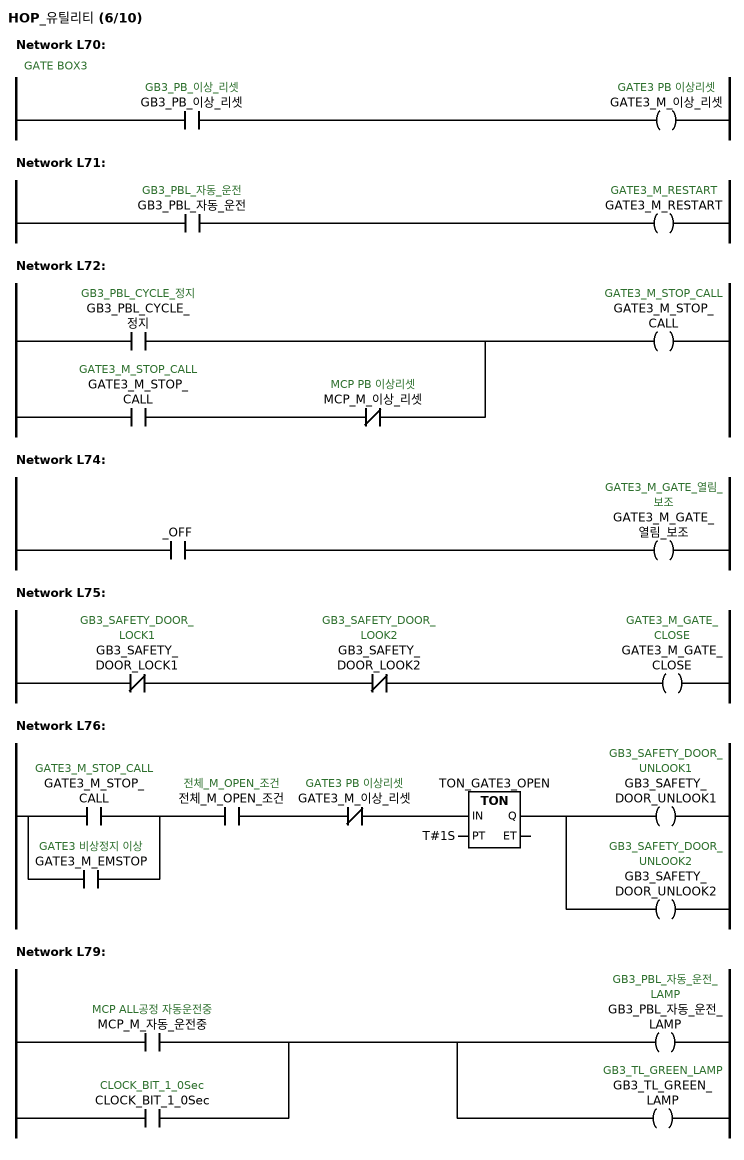
(* GATE BOX3 *)
(* Rung L70 *)
GATE3_M_이상_리셋 := GB3_PB_이상_리셋;
(* Rung L71 *)
GATE3_M_RESTART := GB3_PBL_자동_운전;
(* Rung L72 *)
GATE3_M_STOP_CALL := GB3_PBL_CYCLE_정지 OR (GATE3_M_STOP_CALL AND NOT MCP_M_이상_리셋);
(* Rung L74 *)
GATE3_M_GATE_열림_보조 := _OFF;
(* Rung L75 *)
GATE3_M_GATE_CLOSE := NOT GB3_SAFETY_DOOR_LOCK1 AND NOT GB3_SAFETY_DOOR_LOOK2;
(* Rung L76 *)
TON_GATE3_OPEN(IN := (GATE3_M_STOP_CALL OR GATE3_M_EMSTOP) AND 전체_M_OPEN_조건 AND NOT GATE3_M_이상_리셋, PT := T#1S);
GB3_SAFETY_DOOR_UNLOOK1 := TON_GATE3_OPEN.Q;
GB3_SAFETY_DOOR_UNLOOK2 := TON_GATE3_OPEN.Q;
(* Rung L79 *)
GB3_PBL_자동_운전_LAMP := MCP_M_자동_운전중 OR CLOCK_BIT_1_0Sec;
GB3_TL_GREEN_LAMP := MCP_M_자동_운전중 OR CLOCK_BIT_1_0Sec;

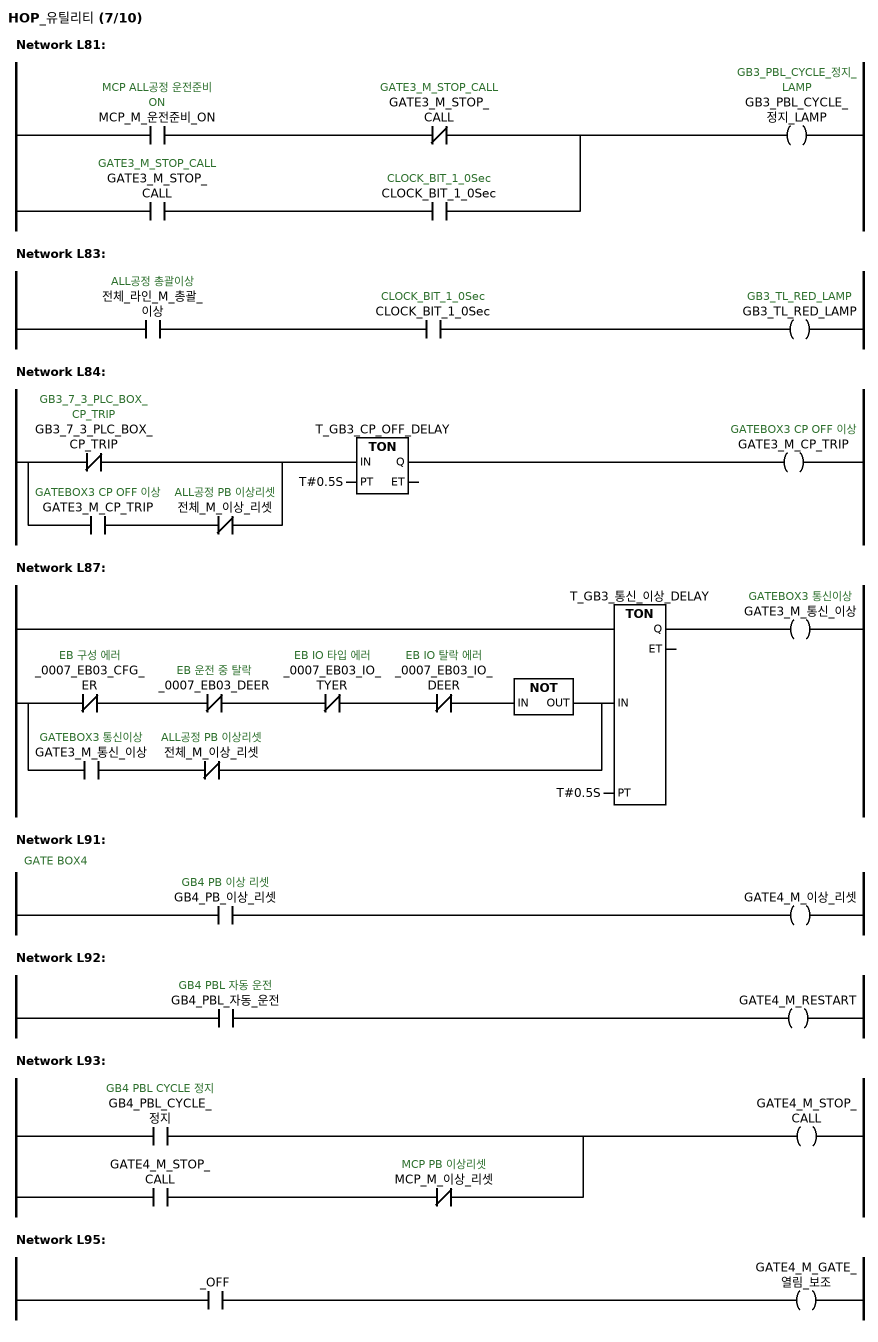
(* Rung L81 *)
GB3_PBL_CYCLE_정지_LAMP := (MCP_M_운전준비_ON AND NOT GATE3_M_STOP_CALL) OR (GATE3_M_STOP_CALL AND CLOCK_BIT_1_0Sec);
(* Rung L83 *)
GB3_TL_RED_LAMP := 전체_라인_M_총괄_이상 AND CLOCK_BIT_1_0Sec;
(* Rung L84 *)
T_GB3_CP_OFF_DELAY(IN := NOT GB3_7_3_PLC_BOX_CP_TRIP OR (GATE3_M_CP_TRIP AND NOT 전체_M_이상_리셋), PT := T#0.5S);
GATE3_M_CP_TRIP := T_GB3_CP_OFF_DELAY.Q;
(* Rung L87 *)
T_GB3_통신_이상_DELAY(IN := (NOT (NOT _0007_EB03_CFG_ER AND NOT _0007_EB03_DEER AND NOT _0007_EB03_IO_TYER AND NOT _0007_EB03_IO_DEER)) OR (GATE3_M_통신_이상 AND NOT 전체_M_이상_리셋), PT := T#0.5S);
GATE3_M_통신_이상 := T_GB3_통신_이상_DELAY.Q;
(* GATE BOX4 *)
(* Rung L91 *)
GATE4_M_이상_리셋 := GB4_PB_이상_리셋;
(* Rung L92 *)
GATE4_M_RESTART := GB4_PBL_자동_운전;
(* Rung L93 *)
GATE4_M_STOP_CALL := GB4_PBL_CYCLE_정지 OR (GATE4_M_STOP_CALL AND NOT MCP_M_이상_리셋);
(* Rung L95 *)
GATE4_M_GATE_열림_보조 := _OFF;

